{attribute 'monitoring':='call'}
PROPERTY MoversInZone : REFERENCE TO ARRAY [0..(CHALET_BaseComponents.BaseParameterlist.MAX_OBJECTS-1)] OF I_XP_Mover_PLC // Return a sorted list of movers in this zone. Index 0 is the mover in Front.
GET
END_GET
END_PROPERTY

END_INTERFACE

// COMPONENTs/Path/FB_XP_Path
{attribute 'enable_dynamic_creation'}
{attribute 'no_explicit_call' := 'Do not call the body - Stick to OOP'}
FUNCTION_BLOCK FB_XP_Path EXTENDS FB_CH_Object IMPLEMENTS I_XP_Path
VAR
	fbTracksUsed : FB_CH_List;
	ipStartStation, ipDestinationStation : I_XP_Station;
	fPathLength : LREAL;
END_VAR

METHOD DistanceToDestiantion : LREAL
VAR_INPUT
	ipTrack : I_XP_Track;
	fPosOnTrack : LREAL;
END_VAR
VAR
	bCorrectPos, bCorrectTrack : BOOL;
	bPosFound : BOOL;
	fDistReturnNotOnThisTrack : LREAL;
	fStart, fEnd : LREAL;
	ipEachTrack : I_XP_Track; 
END_VAR
VAR
	//Todo add tolerance to Size >1
	fToleranceWindow : LREAL := 0.001;//[mm] if Mover is this distance mor far away from the parent, return 0mm
END_VAR
IF ipTrack = 0 THEN
	//Error -  invalide interface
	DistanceToDestiantion := CHALET_BaseComponents.GVL_Datatypes.cMaxLreal;
	RETURN;
END_IF

fDistReturnNotOnThisTrack := CHALET_BaseComponents.GVL_Datatypes.cMaxLreal;

IF (fbTracksUsed.OIDInList(ipTrack.OID) = 0) OR fPosOnTrack < 0 OR  fPosOnTrack > ipTrack.Length THEN
	//Error -  position not on track
	DistanceToDestiantion := fDistReturnNotOnThisTrack;
	RETURN;
END_IF


IF fbTracksUsed.Size = 1 THEN
	bCorrectPos := F_InLimitTest(fMinimum :=  THIS^.StationStart.PositionOnTrack, fInput:=fPosOnTrack , fMaximum:=  (THIS^.StationDestination.PositionOnTrack + fToleranceWindow));
	bCorrectTrack := (ipTrack = StationDestination.AccocietedTrack);

	IF bCorrectPos AND bCorrectTrack THEN
		DistanceToDestiantion := F_GetDistToPosModulo(fTargetPosition := THIS^.StationDestination.PositionOnTrack, fActualPosition := fPosOnTrack, fModulo := ipTrack.Length);
		//check tolerance window
		IF (DistanceToDestiantion + fToleranceWindow) >= ipTrack.Length THEN
			DistanceToDestiantion := 0.0;
		END_IF
	ELSE
		DistanceToDestiantion := fDistReturnNotOnThisTrack;
	END_IF
	RETURN;
END_IF


IF fbTracksUsed.Size > 1 THEN 
	fbTracksUsed.ResetIterator();	
	
	////First track in list
	IF ToXpTrack(fbTracksUsed.GetNextObject(),ipEachTrack) THEN
		fStart 	:= THIS^.StationStart.PositionOnTrack;
		fEnd 	:= ipEachTrack.Length;
		
		bCorrectPos := F_InLimitTest(fMinimum :=  fStart, fInput:=fPosOnTrack , fMaximum:=  fEnd);
		bCorrectTrack := (ipTrack = ipEachTrack);
		IF bCorrectPos AND bCorrectTrack THEN
			bPosFound := TRUE;
			DistanceToDestiantion := fEnd - fPosOnTrack;
		END_IF
	END_IF
	
	
	//All tracks in between
	WHILE fbTracksUsed.HasNextObject() DO
		IF ToXpTrack(fbTracksUsed.GetNextObject(),ipEachTrack) AND_THEN fbTracksUsed.HasNextObject() THEN
			fStart 	:= 0;
			fEnd 	:= ipEachTrack.Length;
			
			// still locking for the startpoint to measure the distance to Destination
			IF NOT bPosFound THEN
				bCorrectPos := F_InLimitTest(fMinimum :=  fStart, fInput:=fPosOnTrack , fMaximum:=  fEnd);
				bCorrectTrack := (ipTrack = ipEachTrack);
				IF bCorrectPos AND bCorrectTrack THEN
					bPosFound := TRUE;
					DistanceToDestiantion := fEnd - fPosOnTrack;
				END_IF
			ELSE
				// add all the tracklengths
				DistanceToDestiantion := DistanceToDestiantion + fEnd;		
			END_IF
		END_IF
	END_WHILE	
	
	
	//Last track
		fStart 	:= 0;
		fEnd 	:= (THIS^.StationDestination.PositionOnTrack + fToleranceWindow);
		// still locking for the startpoint to measure the distance to Destination
		IF NOT bPosFound THEN
			bCorrectPos := F_InLimitTest(fMinimum :=  fStart, fInput:=fPosOnTrack , fMaximum :=  fEnd);
			bCorrectTrack := (ipTrack = ipEachTrack);
			IF bCorrectPos AND bCorrectTrack THEN
				bPosFound := TRUE;
				DistanceToDestiantion := MAX(0, THIS^.StationDestination.PositionOnTrack - fPosOnTrack);
			END_IF
		ELSE
			// add all the tracklengths
			DistanceToDestiantion := DistanceToDestiantion + fEnd;		
		END_IF

	
	fbTracksUsed.RestoreIterator();
	
	IF NOT bPosFound THEN
		DistanceToDestiantion := fDistReturnNotOnThisTrack;
		RETURN;
	END_IF
END_IF
END_METHOD

{attribute 'monitoring':='call'}
//[mm]
PROPERTY Length : LREAL
GET
Length := THIS^.fPathLength;
END_GET
SET
THIS^.fPathLength := Length;
END_SET
END_PROPERTY

{attribute 'monitoring':='call'}
PROPERTY LUID : STRING //Locally unique identifier
GET
VAR
	sTempName : STRING;
END_VAR
IF ipStartStation <> 0 AND ipDestinationStation <> 0 THEN
	sTempName := CONCAT(sTempName, ipStartStation.LUID);
	sTempName := CONCAT(sTempName, ' to ' );
	sTempName := CONCAT(sTempName, ipDestinationStation.LUID);
	
ELSIF ipStartStation <> 0 THEN
	sTempName := CONCAT(sTempName, ipStartStation.LUID);
	sTempName := CONCAT(sTempName, ' to ?' );

ELSIF ipDestinationStation <> 0 THEN
	sTempName := CONCAT(sTempName, '? to ' );
	sTempName := CONCAT(sTempName, ipDestinationStation.LUID);
	
ELSE 
	sTempName := ' Unknown path';
END_IF


LUID := sTempName;
END_GET
END_PROPERTY

{attribute 'monitoring':='call'}
PROPERTY StationDestination : I_XP_Station
GET
StationDestination := THIS^.ipDestinationStation;
END_GET
SET
THIS^.ipDestinationStation := StationDestination;
END_SET
END_PROPERTY

{attribute 'monitoring':='call'}
PROPERTY StationStart  : I_XP_Station
GET
StationStart := THIS^.ipStartStation;
END_GET
SET
THIS^.ipStartStation := StationStart;
END_SET
END_PROPERTY

{attribute 'monitoring':='call'}
//List of tracks
PROPERTY TracksUsed : REFERENCE TO FB_CH_List
GET
TracksUsed REF= THIS^.fbTracksUsed;
END_GET
END_PROPERTY

END_FUNCTION_BLOCK

// FUNCTIONs/F_InLimitTest
FUNCTION F_InLimitTest : BOOL
VAR_INPUT
	fMinimum 	: LREAL;
	fMaximum 	: LREAL;
	fInput 		: LREAL;
END_VAR

//Normal case
// 9 Max
// 5 Test
// 1 Min
IF fMinimum <= fMaximum THEN
	F_InLimitTest := (fInput >= fMinimum) AND (fInput <= fMaximum);
	
//Modulo case	
// 6 | 6  Max
// 5 | 9  Test
// 8 | 8  Min
ELSIF fMinimum > fMaximum THEN
	F_InLimitTest := NOT((fInput > fMaximum) AND (fInput < fMinimum));
END_IF

END_FUNCTION

// FUNCTIONs/F_GetDistToPosModulo
FUNCTION F_GetDistToPosModulo : LREAL //This is only working in Positiv Direktion
VAR_INPUT
	fTargetPosition : LREAL;
	fActualPosition : LREAL;
	fModulo 		: LREAL;
END_VAR

VAR

END_VAR

IF fTargetPosition < fActualPosition THEN
	fTargetPosition := fTargetPosition + fModulo;
END_IF

F_GetDistToPosModulo := fTargetPosition - fActualPosition;

END_FUNCTION

// COMPONENTs/Stationen/A-Star-Node/FB_AStarNode
FUNCTION_BLOCK FB_AStarNode EXTENDS FB_CH_Object IMPLEMENTS I_PathAStarNode
VAR
	{attribute 'hide'}  
	ipStation : I_XP_Station;
	{attribute 'hide'}  
	fbRouteUsedToNode : FB_CH_LIST;	
END_VAR

{attribute 'monitoring':='call'}
PROPERTY LUID : STRING
GET
IF THIS^.Station <> 0 THEN
	LUID := THIS^.Station.LUID;
END_IF
END_GET
END_PROPERTY

{attribute 'monitoring':='call'}
PROPERTY PathLength : LREAL
GET
VAR
	ipEachPath : I_XP_Path;
END_VAR
PathLength := 0.0;


fbRouteUsedToNode.ResetIterator();
WHILE fbRouteUsedToNode.HasNextObject() DO
	IF __QUERYINTERFACE(fbRouteUsedToNode.GetNextObject(), ipEachPath) THEN
		PathLength := PathLength + ipEachPath.Length;
	END_IF
END_WHILE
fbRouteUsedToNode.RestoreIterator();
END_GET
END_PROPERTY

{attribute 'monitoring':='call'}
PROPERTY RouteUsedToNode : REFERENCE TO FB_CH_List
GET
RouteUsedToNode REF= fbRouteUsedToNode;
END_GET
END_PROPERTY

//here in this case the SortOrder is used to get the shortest path. 
PROPERTY SortOrderInList : UDINT
GET
SortOrderInList := TO_UDINT(THIS^.PathLength);
END_GET
END_PROPERTY

{attribute 'monitoring':='call'}
PROPERTY Station : I_XP_Station
GET
Station := ipStation;
END_GET
SET
ipStation := Station;
END_SET
END_PROPERTY

END_FUNCTION_BLOCK

// COMPONENTs/Stationen/A-Star-Node/I_PathAStarNode
INTERFACE I_PathAStarNode EXTENDS I_CH_Object

{attribute 'monitoring':='call'}
PROPERTY PathLength : LREAL
GET
END_GET
END_PROPERTY

{attribute 'monitoring':='call'}
PROPERTY RouteUsedToNode : REFERENCE TO FB_CH_List
GET
END_GET
END_PROPERTY

{attribute 'monitoring':='call'}
PROPERTY Station : I_XP_Station
GET
END_GET
SET
END_SET
END_PROPERTY

END_INTERFACE

// COMPONENTs/Stationen/FB_XP_Station
{attribute 'enable_dynamic_creation'}
{attribute 'no_explicit_call' := 'Do not call the body - Stick to OOP'}
(* XPlanar station - n per associated XPlanar. Can be instantiated as an array and/or individually
	The stations are the main component of the application. As soon as the system has been started up and all movers are on the track, the movers are only sent from one station to the next.
	Parameters:
		xPos, yPos 			= Absolute position of the station on the xPlanar.
		ipAccocietedTrack 	= The track on which the station is located. If the XY position is not on this track, the next possible track position is assumed on this track.
		sUniqueName 		= Unique name that may only exist once.
		sTargetGroup 		= A name for a group to which this station belongs. Important for redundant stations
 *)	
FUNCTION_BLOCK FB_XP_Station EXTENDS FB_CH_Object IMPLEMENTS I_XP_Station, I_XP_Station_PLC
VAR
	//optional - To visualize the station position in LiveView
	fbOptionalTrackUsedInLiveView : MC_PlanarTrack;

	{attribute 'hide'}
	bErrorDuringFbInit : BOOL;	//Fatal error - Not possible to reset
	
	{attribute 'hide'}
	bInitDone : BOOL;
	{attribute 'hide'}	
	bTrackIsSetInFbInit : BOOL;
	{attribute 'hide'}	
	bMoversInPlace : BOOL;
	{attribute 'hide'}                   	
	eActiveCommand 		: CHALET_Nc.E_NcAxisCommands := CHALET_Nc.E_NcAxisCommands.None;
	{attribute 'hide'}	
	ipXpSystem : I_XP_System_Registration;
	{attribute 'hide'}
	bReadyToRecvMovers 		: BOOL := TRUE;
	{attribute 'hide'}
	nCtsMoversMustLeaveThisStation : UDINT;
	{attribute 'hide'}
	sTargetGroup 				: STRING;
	
	{attribute 'hide'}
	bSuppressDynamicsChange		: BOOL; // Suppress to change the dynamic(Gap+velocity) of passing movers. This is usefull in startup
	{attribute 'hide'}
	fMoverGapAtExit 			: LREAL := XPlanarParameterlist.F_GAP_DEFAULT; // Every mover that leaves or passes the station gets this new gap as a target.
	{attribute 'hide'}	
	fbPositionPlanned : PositionXY; //this is the configured/planned position of the station. set via FB_init. If it is not on the track, the PosOnTrackXY is different
	{attribute 'hide'}	
	fPositionOnTrack : LREAL;
	{attribute 'hide'}
	fbPositionOnTrackXY : PositionXY;	
	{attribute 'hide'}	
	nState_Configuring: INT;
	{attribute 'hide'}	
	ipAccocietedTrack : I_XP_Track;
	{attribute 'hide'}
	nMoverQueueSize 			: UINT;
	{attribute 'hide'}
	fTargetPosWindow			: LREAL := 0.05; //[mm]
	{attribute 'hide'}
	tTargetPosMonitoringTime	: TIME := T#0MS;

	
	(*List of stations*)
	{attribute 'hide'}	
	fbStationsAhead : FB_CH_List;
	{attribute 'hide'}	
	fbStationsBehinde : FB_CH_List;
	
	(*List of paths*)
	{attribute 'hide'}	
	fbListPathAhead : FB_CH_List;
	{attribute 'hide'}
	fbListPathBehind : FB_CH_List;
	
	(* Lists to handle the ownership of movers *)
	{attribute 'hide'}
	fbAssignedMovers 			: FB_CH_List;		// Movers approaching the station. This station is the parent of this movers
	{attribute 'hide'}
	fbFeedback : FB_CH_Feedback(ipSourceInfo := fbSourceInfo);		
	
	//Simulation
	{attribute 'hide'}
	fSimulationProcessDuration 	: LREAL; //[s]
	{attribute 'hide'}
	sSimulationTargetStation	: STRING; //GroupID of the target station to automatic send after the duration
	
	
	//ipXpSystem Is Not Valid at this point, call the konstruktor again in the FB_Init
	{attribute 'hide'}
	fbTrigger 					: FB_XP_Trigger(ipXpSystem);
	{attribute 'hide'}
	fbSortedListMoversInQueue	: FB_XP_SoretedListOfMover(	ipXpStation := THIS^,
															ipListOfMoversToCheck := fbAssignedMovers );
	{attribute 'hide'}
	fDecisionDistance: LREAL;//[mm]
	{attribute 'hide'}
	bNetworkHasTrackBranches : BOOL;//True if atleas on branche is existing in network
	{attribute 'hide'}
	sFilter : STRING :=  XPlanarParameterlist.S_ANY_STATION_NAME;
	{attribute 'hide'}	
	fbAlarmStationIsBlocked : FB_TcAlarm;
END_VAR

// Dynamic to use if an Mvoer passes the station
// Every mover that leaves or passes the station gets this new velo as a target.
VAR
	{attribute 'hide'}	
	fMoverVeloAtExit : MC_LREAL := MC_DEFAULT; //equivalent to data type LREAL + MC_DEFAULT, MC_MAXIMUM
	{attribute 'hide'}	
    fMoverAccAtExit : MC_LREAL := MC_DEFAULT; //equivalent to data type LREAL + MC_DEFAULT, MC_MAXIMUM
	{attribute 'hide'}	
    fMoverDecAtExit : MC_LREAL := MC_DEFAULT; //equivalent to data type LREAL + MC_DEFAULT, MC_MAXIMUM
END_VAR

METHOD PROTECTED CheckInvalideParameter : HRESULT
VAR
 	ipStation : I_XP_Station;
	fbListOfStationsToCheck : FB_CH_List;
END_VAR
VAR_INST
	{attribute 'hide'}	
	fbAlarm : FB_TcAlarm;
END_VAR
//Get a list of all station whitout this station
fbListOfStationsToCheck.Duplicate(THIS^.ipXpSystem.StationsUsed);
fbListOfStationsToCheck.RemoveObject(THIS^);


fbListOfStationsToCheck.ResetIterator();
WHILE fbListOfStationsToCheck.HasNextObject() DO
	IF ToXpStation(fbListOfStationsToCheck.GetNextObject(), ipStation) THEN
		
		//Check for same positions
		IF (ipStation.PositionOnTrack = THIS^.PositionOnTrack) AND (ipStation.AccocietedTrack = THIS^.AccocietedTrack)  THEN
			//Error two stations have same position on track
			CheckInvalideParameter := E_FAIL;
			IF NOT fbAlarm.bRaised THEN
				fbAlarm.CreateEx(stEventEntry:=TC_EVENTS.CHALET_XPlanar_Events.DuplicateStationPositions, ipSourceInfo := THIS^.fbSourceInfo, bWithConfirmation := FALSE);
				fbAlarm.ipArguments.AddStringByValue(THIS^.LUID).AddStringByValue(ipStation.LUID);
				fbAlarm.Raise(0);			
			END_IF
			RETURN;
		END_IF
		
		//Check same unique id
		IF (ipStation.LUID = THIS^.LUID) THEN
			//Error two stations have same unique id
			CheckInvalideParameter := E_FAIL;
			IF NOT fbAlarm.bRaised THEN
				fbAlarm.CreateEx(stEventEntry:=TC_EVENTS.CHALET_XPlanar_Events.DuplicateStationName, ipSourceInfo := THIS^.fbSourceInfo, bWithConfirmation := FALSE);
				fbAlarm.ipArguments.AddStringByValue(THIS^.LUID);
				fbAlarm.Raise(0);			
			END_IF
			RETURN;
		END_IF
		
		fbListOfStationsToCheck.RemoveObject(ipStation);
	END_IF
END_WHILE
END_METHOD

METHOD protected GetAccocietedTrack : HRESULT
VAR
	ipTrack : I_XP_Track;

	fPosOnTrack, fDist	: LREAL;
	fbPositionXYC : PositionXYC;
	fbPositionXY : PositionXY;
	ipClosestTrack : I_XP_Track;
	fDistClosestTrack : LREAL := CHALET_BaseComponents.GVL_Datatypes.cMaxLreal;
END_VAR
//If track is not defind during FB_init, get closest track 
IF NOT bTrackIsSetInFbInit THEN
	THIS^.ipAccocietedTrack := 0;
	THIS^.ipXpSystem.Tracks.ResetIterator();
	WHILE THIS^.ipXpSystem.Tracks.HasNextObject() DO
		IF ToXpTrack(THIS^.ipXpSystem.Tracks.GetNextObject(),ipTrack) THEN 
			
			fPosOnTrack := ipTrack.PlanarTrack.GetArcLengthClosestTo(geometry:= THIS^.fbPositionPlanned);
			//Get the XYC Pos on track
			ipTrack.PlanarTrack.GetPositionAt(fPosOnTrack, fbPositionXYC);
			//Get radius/ distance to positionTarget
			fbPositionXY.x  := THIS^.fbPositionPlanned.x - fbPositionXYC.x;
			fbPositionXY.y  := THIS^.fbPositionPlanned.y - fbPositionXYC.y;
			fDist := fbPositionXY.GetRadius();
			
			IF fDist < fDistClosestTrack THEN
				fDistClosestTrack := fDist;
				ipClosestTrack := ipTrack;
			END_IF
		END_IF
	END_WHILE
	THIS^.ipXpSystem.Tracks.RestoreIterator();
	
	
	THIS^.ipAccocietedTrack := ipClosestTrack;	
END_IF

// Error - No track found
IF THIS^.ipAccocietedTrack = 0 THEN
	GetAccocietedTrack := E_FAIL;
	RETURN;
END_IF
END_METHOD

METHOD GetDecisionDistance : HRESULT
VAR
	fDistToStartOfTrack : LREAL := CHALET_BaseComponents.GVL_Datatypes.cMaxLreal;
	fDistStationBehind : LREAL := CHALET_BaseComponents.GVL_Datatypes.cMaxLreal;
	
	ipPath : I_XP_Path;
END_VAR
(*
As soon as the mover is closer than this distance, the mover can be sent on to the next one if necessary.
This is the distance from the station to the end of the track or the shortest path to this station. Depending on which is closer. This is to ensure that the mover can no longer be overhauled.
*)
fDistToStartOfTrack := THIS^.PositionOnTrack;

THIS^.PathsBehinde.ResetIterator();
WHILE THIS^.PathsBehinde.HasNextObject() DO
	IF __QUERYINTERFACE(THIS^.PathsBehinde.GetNextObject(), ipPath) THEN
		fDistStationBehind := MIN(fDistStationBehind, ipPath.Length);
	END_IF
END_WHILE
THIS^.PathsBehinde.RestoreIterator();

THIS^.fDecisionDistance := CHALET_BaseComponents.GVL_Datatypes.cMaxLreal;
THIS^.fDecisionDistance := MIN(THIS^.fDecisionDistance, (fDistToStartOfTrack - 1.0));
THIS^.fDecisionDistance := MIN(THIS^.fDecisionDistance, (fDistStationBehind - 1.0));
THIS^.fDecisionDistance := MIN(THIS^.fDecisionDistance, XPlanarParameterlist.F_DIST_SET_NEW_MOVE_CMD_BEFORE_REACHING_PARENT_STATION);


IF THIS^.fDecisionDistance < 1.0 THEN 
	THIS^.fDecisionDistance := 1.0;
END_IF

GetDecisionDistance := S_OK;
END_METHOD

METHOD protected GetPathsAhead : HRESULT
VAR_INPUT
END_VAR

VAR
	fbPathElementsToCheck : FB_CH_List;
	fbListStationsToGetClosest : FB_CH_List;	
	ipObjectPathAhead 				: I_CH_Object;
	ipStation,ipStation1,ipStation2 	: I_XP_Station;
	ipTrack					: I_XP_Track; 
	ipLastAddedTrack 		: I_XP_Track;
	ipPath 					: I_XP_Path;
	ipPathCurrentLoop  		: I_XP_Path;
	
	
	pFbPath, pFbPathCurrentLoop : POINTER TO FB_XP_Path;
	
	fSeachStartPoint : LREAL;
	nIdx : UDINT;
END_VAR
(*
Check whether there is a station further ahead on this track than this one.
If there is no other station on the track, the previous tracks are filled into a list and searched one after the other to see if they have valid stations. 
If the tracks also have no stations, the track before it is added to the list,...
*)

//Clear list, delete dynamic_creation path objects
WHILE NOT fbListPathAhead.IsEmpty DO
	ipObjectPathAhead := fbListPathAhead.GetRandomObject();
	fbListPathAhead.RemoveObject(ipObjectPathAhead);
	
	//get pointer and delete
	IF __QUERYPOINTER(ipObjectPathAhead, pFbPath) THEN
		__DELETE(pFbPath);
	END_IF	
		
END_WHILE


//new dynamic_creation path objects
pFbPath := __NEW(FB_XP_Path);
//init path
pFbPath^.StationStart := THIS^;
pFbPath^.TracksUsed.ResetIterator();
pFbPath^.TracksUsed.AddObject(THIS^.AccocietedTrack);

//add to list
fbPathElementsToCheck.AddObject(pFbPath^);

//On first pathsearch get an Station who is further ahead than this
fSeachStartPoint := THIS^.PositionOnTrack;



//While list is not empty
WHILE NOT fbPathElementsToCheck.IsEmpty DO
	__QUERYINTERFACE(fbPathElementsToCheck.GetRandomObject(), ipPathCurrentLoop);
	__QUERYINTERFACE(ipPathCurrentLoop.TracksUsed.GetNextObject(),ipLastAddedTrack);
	
	
	//Closed loop
	IF ipLastAddedTrack.ClosedLoop THEN
		//on closed-loop add all stations of this track to list
		fbListStationsToGetClosest.Duplicate(ipLastAddedTrack.StationsOnTrack);
	
		//remove THIS station from list if more than on station is existing
		IF fbListStationsToGetClosest.Size > 1 THEN
			fbListStationsToGetClosest.RemoveObject(THIS^);
		END_IF
	
		
	
	ELSE
		//Not closed loop	
		//Get a List of all stations on track Position > Startpoint
		ipLastAddedTrack.StationsOnTrack.ResetIterator();
		fbListStationsToGetClosest.Clear();
		WHILE ipLastAddedTrack.StationsOnTrack.HasNextObject() DO
			IF ToXpStation(ipLastAddedTrack.StationsOnTrack.GetNextObject(),ipStation) THEN
				//Add all station ahead to list. on closed-loop add all stations of this track to list
				IF ipStation.PositionOnTrack > fSeachStartPoint THEN
					fbListStationsToGetClosest.AddObject(ipStation);
				END_IF
			END_IF
		END_WHILE	
	END_IF
		
	

	
	//Get closest to startpos(0mm)
	WHILE fbListStationsToGetClosest.Size > 1 DO
		fbListStationsToGetClosest.ResetIterator();
		__QUERYINTERFACE(fbListStationsToGetClosest.GetNextObject(),ipStation1);
		__QUERYINTERFACE(fbListStationsToGetClosest.GetNextObject(),ipStation2);
		
		//If station1 is closer to start than station2, remove station2
		IF 		F_GetDistToPosModulo(fTargetPosition := ipStation1.PositionOnTrack, fActualPosition := fSeachStartPoint, fModulo := ipLastAddedTrack.Length) 
			< 	F_GetDistToPosModulo(fTargetPosition := ipStation2.PositionOnTrack, fActualPosition := fSeachStartPoint, fModulo := ipLastAddedTrack.Length) THEN
			fbListStationsToGetClosest.RemoveObject(ipStation2);
		ELSE	
			fbListStationsToGetClosest.RemoveObject(ipStation1);
		END_IF
	END_WHILE
	
	
	IF fbListStationsToGetClosest.Size = 1 THEN
		//Station FOUND
		__QUERYINTERFACE(fbListStationsToGetClosest.GetRandomObject(), ipStation);
		ipPathCurrentLoop.StationDestination := ipStation;
		
		//Calculate Tracklentgh
		ipPathCurrentLoop.TracksUsed.ResetIterator();
		WHILE ipPathCurrentLoop.TracksUsed.HasNextObject() DO
			IF ToXpTrack(ipPathCurrentLoop.TracksUsed.GetNextObject(),ipTrack) THEN
				ipPathCurrentLoop.Length := ipPathCurrentLoop.Length + ipTrack.Length;
			END_IF
		END_WHILE	
		ipPathCurrentLoop.Length := ipPathCurrentLoop.Length - ipPathCurrentLoop.StationStart.PositionOnTrack;
		ipPathCurrentLoop.Length := ipPathCurrentLoop.Length - ipPathCurrentLoop.StationDestination.AccocietedTrack.Length + ipPathCurrentLoop.StationDestination.PositionOnTrack;
		
		//Modulo on cloosed track add 1 track length 
		IF ipPathCurrentLoop.StationStart.AccocietedTrack = ipPathCurrentLoop.StationDestination.AccocietedTrack AND 
			ipPathCurrentLoop.StationStart.PositionOnTrack > ipPathCurrentLoop.StationDestination.PositionOnTrack THEN
				ipPathCurrentLoop.Length := ipPathCurrentLoop.Length + ipPathCurrentLoop.StationDestination.AccocietedTrack.Length;
		END_IF
		
		fbListPathAhead.AddObject(ipPathCurrentLoop);
		fbPathElementsToCheck.RemoveObject(ipPathCurrentLoop);
	ELSE
		//Station NOT-FOUND, add the subsequent tracks in the list
		ipLastAddedTrack.TracksAhead.ResetIterator();
		WHILE ipLastAddedTrack.TracksAhead.HasNextObject() DO
			ToXpTrack(ipLastAddedTrack.TracksAhead.GetNextObject(), ipTrack);
			//dublicate current path
			pFbPath := __NEW(FB_XP_Path);
			//Get pointer from fb behinde this interface
			__QUERYPOINTER(ipPathCurrentLoop, pFbPathCurrentLoop);
			MEMCPY(destAddr := pFbPath, srcAddr := pFbPathCurrentLoop, n := SIZEOF(FB_XP_Path));
			//Add the new track to fresh created path
			pFbPath^.TracksUsed.AddObject(ipTrack);
			//Add to list to check
			fbPathElementsToCheck.AddObject(pFbPath^);
			
		END_WHILE

		
		//delete current path
		fbPathElementsToCheck.RemoveObject(ipPathCurrentLoop);

		//get pointer and delete
		IF __QUERYPOINTER(ipPathCurrentLoop, pFbPath) THEN
			__DELETE(pFbPath);
		END_IF	
		
	END_IF

	fSeachStartPoint := -0.1;
END_WHILE
END_METHOD

METHOD protected GetPathsBehind : HRESULT
VAR
	ipThisStation : I_XP_Station;
	ipXpStation : I_XP_Station;
	ipPath		: I_XP_Path;
END_VAR
ipThisStation := THIS^;
fbListPathBehind.Clear();

THIS^.fbStationsBehinde.ResetIterator();
WHILE THIS^.fbStationsBehinde.HasNextObject() DO
	IF __QUERYINTERFACE(THIS^.fbStationsBehinde.GetNextObject(),ipXpStation) THEN
		ipXpStation.PathsAhead.ResetIterator();
		WHILE ipXpStation.PathsAhead.HasNextObject() DO
			IF __QUERYINTERFACE(ipXpStation.PathsAhead.GetNextObject(),ipPath) AND_THEN ipPath.StationDestination = ipThisStation THEN
				//add path to this station to list
				fbListPathBehind.AddObject(ipPath);
			END_IF
		END_WHILE	
	END_IF
END_WHILE
END_METHOD

METHOD PROTECTED GetPosOnTrack : HRESULT
VAR
	fbPositionXYC : PositionXYC;
END_VAR
//GetArcLengthClosestTo track
THIS^.fPositionOnTrack := THIS^.ipAccocietedTrack.PlanarTrack.GetArcLengthClosestTo(geometry:= THIS^.fbPositionPlanned);

//Get the XYC Pos on track
THIS^.ipAccocietedTrack.PlanarTrack.GetPositionAt(THIS^.PositionOnTrack, fbPositionXYC);

//XYC -> XY
THIS^.fbPositionOnTrackXY.SetValuesXY(fbPositionXYC.x,fbPositionXYC.y);


//Check for NaN
IF NOT(THIS^.fPositionOnTrack = THIS^.fPositionOnTrack) THEN
	GetPosOnTrack := E_FAIL;
	RETURN;
END_IF
END_METHOD

METHOD PROTECTED GetStationAhead : HRESULT
VAR
	ipPath 		: I_XP_Path;
END_VAR
fbStationsAhead.Clear();


fbListPathAhead.ResetIterator();
WHILE fbListPathAhead.HasNextObject() DO
	IF __QUERYINTERFACE(fbListPathAhead.GetNextObject(),ipPath) THEN
		//add StationDestination to list
		fbStationsAhead.AddObject(ipPath.StationDestination);
	END_IF
END_WHILE
END_METHOD

METHOD PROTECTED GetStationBehinde : HRESULT
VAR_INPUT
END_VAR
VAR
	ipThisStation : I_XP_Station;
	ipXpStation : I_XP_Station;
	ipXpStationAhead : I_XP_Station;
END_VAR
ipThisStation := THIS^;
fbStationsBehinde.Clear();

//Check each Station
THIS^.ipXpSystem.StationsUsed.ResetIterator();
WHILE THIS^.ipXpSystem.StationsUsed.HasNextObject() DO
	IF __QUERYINTERFACE(THIS^.ipXpSystem.StationsUsed.GetNextObject(),ipXpStation) THEN
		//check the list of stations ahead if this station one is existing
		ipXpStation.StationsAhead.ResetIterator();
		WHILE ipXpStation.StationsAhead.HasNextObject() DO
			IF __QUERYINTERFACE(ipXpStation.StationsAhead.GetNextObject(),ipXpStationAhead) AND_THEN (ipXpStationAhead = ipThisStation) THEN
				//add station to list
				fbStationsBehinde.AddObject(ipXpStation);
			END_IF
		END_WHILE	
	END_IF
END_WHILE	
THIS^.ipXpSystem.StationsUsed.RestoreIterator();
END_METHOD

METHOD PROTECTED ManageAutomaticallyGeneratedStations : HRESULT
VAR
	ipThisStation : I_XP_Station := THIS^;
	ipTempTrackAhead : I_XP_Track;
	bThisStationIsCreatedAutomatically : BOOL;
	
	bOtherStationsOnThisTrack : BOOL;
	bAnotherTrackAhed : BOOL;
	
	pfbListAllUsedStations : POINTER TO FB_CH_List;
END_VAR
// Check if this station was created by the user, e.g., as a process station, or if it was created automatically at the end of the track to improve track management.
bThisStationIsCreatedAutomatically := (ipThisStation = THIS^.AccocietedTrack.HelperStationAtEndOfTrack);

// Only check automaticali created stations
IF NOT bThisStationIsCreatedAutomatically THEN
	ManageAutomaticallyGeneratedStations := S_OK;
	RETURN;
END_IF



//Set position of this automatic generated station to the end of the accocieted Track
THIS^.PositionXY.x := THIS^.AccocietedTrack.EndPosition.x;
THIS^.PositionXY.y := THIS^.AccocietedTrack.EndPosition.y;



//Check if other Stations are existiong on this track
IF THIS^.AccocietedTrack.StationsOnTrack.Size > 1 THEN
	bOtherStationsOnThisTrack := TRUE;
END_IF

//Another track is before this accocieted track. But the track in front of me is only allowed to have this one track in behind of it.
__QUERYINTERFACE(THIS^.AccocietedTrack.TracksAhead.GetRandomObject(), ipTempTrackAhead);
IF ipTempTrackAhead <> 0 AND_THEN ipTempTrackAhead.TracksBehinde.Size = 1 THEN
	bAnotherTrackAhed := TRUE;
END_IF

//Remove this station from list
/// Todo remove Querypointer - not very OOP
IF (bOtherStationsOnThisTrack OR bAnotherTrackAhed OR NOT XPlanarParameterlist.B_AUTOMATIC_GENARATE_HELPER_STATIONS ) AND __QUERYPOINTER(THIS^.ipXpSystem.StationsUsed, pfbListAllUsedStations) THEN
	//Remove single trackpoint if station is not used
	THIS^.fbOptionalTrackUsedInLiveView.Clear(0);
	pfbListAllUsedStations^.RemoveObject(THIS^);
END_IF
END_METHOD

METHOD SetTrackObjName : HRESULT
VAR
	ipComObject : ITComObject;
	sName : STRING;
END_VAR
FW_ObjMgr_GetObjectInstance(oid:= THIS^.fbOptionalTrackUsedInLiveView.MCTOPLC_STD.TrackOID, iid:= TC_GLOBAL_IID_LIST.IID_ITComObject, pipUnk:= ADR(ipComObject));
IF ipComObject <> 0 THEN
	sName := THIS^.LUID;
	ipComObject.TcSetObjectName(ADR(sName));
	FW_SafeRelease(ADR(ipComObject));
END_IF
END_METHOD

//Call this Methode whith seq 0->99, and wait each step until S_OK is returned
METHOD Configure : HRESULT
VAR_INPUT
	nSeq : UINT; //0->100
END_VAR

VAR_INST
	{attribute 'hide'}
	fbFeedback : MC_PlanarFeedback;	
END_VAR
VAR
	bOptionalTrackUsedInLiveViewIsMapped : BOOL;
	fbPositionXYC : PositionXYC;
	ipEachTrack : I_XP_Track;
END_VAR
bOptionalTrackUsedInLiveViewIsMapped := fbOptionalTrackUsedInLiveView.MCTOPLC_STD.TrackOID <> 0;

CASE nSeq OF
	5:	//Get interface of trackobject
		Configure := THIS^.GetAccocietedTrack();	

	10: //Get closest XY-Position on track
		Configure := THIS^.GetPosOnTrack();
		
	11:	//Automatic add/remove this station from list of all station if it is createt automatic at the end of each track and is (not) used	
		Configure := THIS^.ManageAutomaticallyGeneratedStations();
		
	12: //Check id is unique and not multiple stations at same position
		Configure := THIS^.CheckInvalideParameter();		
				
	13:	//Init Tigger
		fbTrigger.AccocietedTrack := THIS^.AccocietedTrack;
		fbTrigger.PositionOnTrack := THIS^.PositionOnTrack;
		fbTrigger.ListOfMoversToCheck := THIS^.ipXpSystem.MoversPresent;//All mover
		fbTrigger.TriggerDirection := Tc3_Mc3Definitions. MC_DIRECTION.mcDirectionPositive;
		Configure := fbTrigger.Initialize();
	
	14:	//Init Zone		
		Configure := fbSortedListMoversInQueue.Initialize();	
	
	20: //Fill the list of all paths before this station
		Configure := THIS^.GetPathsAhead();		
		
	25: //Fill the list of all stations before this station
		Configure := THIS^.GetStationAhead();

	30: //Fill the list of all paths behinde this station
		Configure := THIS^.GetStationBehinde();	
			
	35: //Fill the list of all stations behinde this station
		Configure := THIS^.GetPathsBehind();

	40: //Determine the distance from which the station can give a new command to a mover
		Configure := THIS^.GetDecisionDistance();
		

//----------------------------------------------------------------		
//The station can optionally be linked to a track object. this track is then displayed in the live view.
//It takes several cycles to prepare the object
	80: IF bOptionalTrackUsedInLiveViewIsMapped THEN
			fbOptionalTrackUsedInLiveView.Clear(fbFeedback);
		END_IF
		
	81:	//Wait for clearing
		IF bOptionalTrackUsedInLiveViewIsMapped THEN
			IF fbFeedback.Done THEN
				Configure := S_OK;
			ELSIF fbFeedback.Busy THEN
				Configure := S_PENDING;
			ELSIF fbFeedback.Error THEN
				Configure := E_FAIL;
			END_IF	
		END_IF

	82: //Set position 
		IF bOptionalTrackUsedInLiveViewIsMapped THEN
			fbPositionXYC.SetValuesXY(THIS^.PositionOnTrackXY.x, THIS^.PositionOnTrackXY.y);
			fbOptionalTrackUsedInLiveView.AppendPosition(position := fbPositionXYC, commandFeedback:= fbFeedback);	
		END_IF	
	
	83:	//Wait for set position
		IF bOptionalTrackUsedInLiveViewIsMapped THEN
			IF fbFeedback.Done THEN
				Configure := S_OK;
			ELSIF fbFeedback.Busy THEN
				Configure := S_PENDING;
			ELSIF fbFeedback.Error THEN
				Configure := E_FAIL;
			END_IF	
		END_IF
		
	84:	//Set name of "track" to stationsname 
		IF bOptionalTrackUsedInLiveViewIsMapped THEN
 			Configure := SetTrackObjName();
		END_IF
//----------------------------------------------------------------

	90: //Create some internal used variable
		THIS^.bNetworkHasTrackBranches := FALSE;
		THIS^.ipXpSystem.Tracks.ResetIterator();
		WHILE THIS^.ipXpSystem.Tracks.HasNextObject() DO
			IF __QUERYINTERFACE(THIS^.ipXpSystem.Tracks.GetNextObject(), ipEachTrack) AND_THEN (ipEachTrack.TracksAhead.Size > 1) THEN
				THIS^.bNetworkHasTrackBranches := TRUE;
				EXIT;
			END_IF
		END_WHILE
		THIS^.ipXpSystem.Tracks.RestoreIterator();
		
		

	100..CHALET_BaseComponents.GVL_Datatypes.cMaxUint: 
		// 100..MaxUint -> Invalide input
		Configure := E_FAIL;
		
	ELSE 
		//If an step is not defind/used return ok
		Configure := S_OK;
END_CASE


fbOptionalTrackUsedInLiveView.Update();
fbFeedback.Update();
END_METHOD

//This method is called when the system is disabled. Links are deleted as they may no longer be valid
METHOD Disassemble : HRESULT
VAR_INPUT
END_VAR
fbStationsAhead.Clear(); 
fbStationsBehinde.Clear(); 
fbListPathAhead.Clear(); 
fbListPathBehind.Clear(); 

Disassemble := S_OK;
END_METHOD

{attribute 'monitoring':='call'}
PROPERTY CtsEmptySpaceInQueue : UDINT
GET
//Handle UINT Overflow
IF THIS^.fbAssignedMovers.Size >= THIS^.nMoverQueueSize THEN
	CtsEmptySpaceInQueue := 0;
ELSE 
	CtsEmptySpaceInQueue := THIS^.nMoverQueueSize - THIS^.fbAssignedMovers.Size;
END_IF
END_GET
END_PROPERTY

{attribute 'monitoring':='call'}
PROPERTY CtsMoversInQueue : UDINT
GET
CtsMoversInQueue := THIS^.fbAssignedMovers.Size;
END_GET
END_PROPERTY

{attribute 'monitoring':='call'}
PROPERTY MoverAccAtExit : MC_LREAL //[mm/s² on Track] Every mover that leaves or passes the station gets this new acceleration as a target.
GET
MoverAccAtExit := THIS^.fMoverAccAtExit;
END_GET
SET
THIS^.fMoverAccAtExit := MoverAccAtExit;
END_SET
END_PROPERTY

{attribute 'monitoring':='call'}
PROPERTY MoverDecAtExit : MC_LREAL //[mm/s² on Track] Every mover that leaves or passes the station gets this new deceleration as a target.
GET
MoverDecAtExit := THIS^.fMoverDecAtExit;
END_GET
SET
THIS^.fMoverdecAtExit := MoverDecAtExit;
END_SET
END_PROPERTY

{attribute 'monitoring':='call'}
PROPERTY MoverQueueSize : UINT
GET
MoverQueueSize := THIS^.nMoverQueueSize;
END_GET
SET
THIS^.nMoverQueueSize := MoverQueueSize;
END_SET
END_PROPERTY

{attribute 'monitoring':='call'}
PROPERTY MoversInPlace : BOOL
GET
THIS^.Prepare();//Prepare time-critical information, if not already done


MoversInPlace := bMoversInPlace;
END_GET
END_PROPERTY

{attribute 'monitoring':='call'}
// Return a sorted list of movers in this zone. Index 0 is the mover in Front
PROPERTY MoversInQueue : REFERENCE TO ARRAY [0..(CHALET_BaseComponents.BaseParameterlist.MAX_OBJECTS-1)] OF I_XP_Mover_PLC
GET
MoversInQueue REF= THIS^.fbSortedListMoversInQueue.MoversInZone;
END_GET
END_PROPERTY

{attribute 'monitoring':='call'}
PROPERTY MoverVelocityAtExit : MC_LREAL //[mm/s on Track] Every mover that leaves or passes the station gets this new velocity as a target.
GET
MoverVelocityAtExit := THIS^.fMoverVeloAtExit;
END_GET
SET
THIS^.fMoverVeloAtExit := MoverVelocityAtExit;
END_SET
END_PROPERTY

METHOD PROTECTED OnMoverPasses : BOOL //This methode is called automaticly from the station and detect mover who is passing the station whitout be in queue.
VAR_INPUT
	ipMoverPasses : I_XP_Mover;
END_VAR
VAR
	ipThisStation : I_XP_Station := THIS^;
	
	//this raises an error 33155 "Target position is not reachable. There is no path available to the target position or target position is unreachable in general."
	bPreventMoveCmdToMoversCurrentPos : BOOL;
END_VAR
IF ipMoverPasses = 0 THEN
	RETURN;
END_IF


//Detect mover who is passing the station whitout be in queue. 
//Adjust to new Dynamics
IF NOT THIS^.bSuppressDynamicsChange AND XPlanarParameterlist.B_STATIONS_OVERRIDE_MOVER_DYN_CONSTRAINT THEN
	//Only if not in this queue
	IF ipMoverPasses.ParentStation <> ipThisStation  THEN
		ipMoverPasses.SetDynConstraint_Path(	V:= THIS^.fMoverVeloAtExit, 
												A:= THIS^.fMoverAccAtExit,
												D:= THIS^.fMoverDecAtExit,
												J:= MC_DEFAULT);
	END_IF
END_IF	



//Detect mover who is passing the station whitout be in queue. 
//Adjust to new Gap
IF NOT THIS^.bSuppressDynamicsChange THEN
	bPreventMoveCmdToMoversCurrentPos := (ipMoverPasses.PositionOnTrack = ipMoverPasses.LastCmdTargetPosition) AND (ipMoverPasses.CurrentTrack = ipMoverPasses.LastCmdTargetTrack);
	//Only if not in this queue
	IF ipMoverPasses.ParentStation <> ipThisStation AND NOT bPreventMoveCmdToMoversCurrentPos THEN
		ipMoverPasses.MoveOnTrack(ipTrack	:= ipMoverPasses.LastCmdTargetTrack,
								fPosition	:= ipMoverPasses.LastCmdTargetPosition, 
								fGap		:= THIS^.fMoverGapAtExit);
	END_IF
END_IF
END_METHOD

//The movers currently in this station must leave the station. 
//The movers actively search for a destination, but only leave if a new destination is available.
METHOD PushMoversOutOfStation : HRESULT
VAR_INPUT
END_VAR
THIS^.nCtsMoversMustLeaveThisStation := THIS^.CtsMoversInQueue;
END_METHOD

{attribute 'monitoring':='call'}
//prevent further movers from entering the station, 
//e.g. to prevent a collision. All movers that are already moving to reach this station will be stopped with a stop 
//and restarted with Ready True.
PROPERTY ReadyToRecvMovers : BOOL
GET
ReadyToRecvMovers := bReadyToRecvMovers;
END_GET
SET
VAR
	ipEachMover : I_XP_Mover;
END_VAR
(* zzz Todo braucht es das?
//Change to Not Ready:
IF (ReadyToRecvMovers = FALSE) AND (bReadyToRecvMovers <> ReadyToRecvMovers) THEN
	//halt all movers on the way
	fbAssignedMovers.ResetIterator();
	WHILE fbAssignedMovers.HasNextObject() DO
		IF ToXpMover(fbAssignedMovers.GetNextObject(),ipEachMover) THEN
			ipEachMover.Halt();	
		END_IF	
	END_WHILE
END_IF

//Change to Ready:
IF (ReadyToRecvMovers = TRUE) AND (bReadyToRecvMovers <> ReadyToRecvMovers) THEN
	//all movers that are on the way have probably been stopped before. when reactivated, the last move command is sent again.
	fbAssignedMovers.ResetIterator();
	WHILE fbAssignedMovers.HasNextObject() DO
		IF ToXpMover(fbAssignedMovers.GetNextObject(),ipEachMover) THEN
			ipEachMover.MoveOnTrack(ipTrack 	:= ipEachMover.LastCmdTargetTrack ,
									fPosition	:= ipEachMover.LastCmdTargetPosition,
									fGap		:= ipEachMover.LastCmdTargetGap);
		END_IF	
	END_WHILE
END_IF
*)
//Store new status
bReadyToRecvMovers := ReadyToRecvMovers;
END_SET
END_PROPERTY

METHOD SendMoversToStation : I_CH_Feedback //All movers in the station are sent to this destination
VAR_INPUT
	sTargetStation: STRING;//unique station name or group of stations
END_VAR
VAR
	nIdx : UDINT;
	ipXpMover : I_XP_Mover;
END_VAR
IF THIS^.fbFeedback.Error THEN
	//Error active/not ready
	THIS^.fbFeedback.LastCommandAccepted	:= FALSE;
	RETURN;
END_IF


//Invalide target
IF sTargetStation = '' THEN
	THIS^.fbFeedback.LastCommandAccepted	:= FALSE;
	RETURN;
END_IF


//Send all Queued movers away by changing the target station destination
THIS^.fbAssignedMovers.ResetIterator();
WHILE THIS^.fbAssignedMovers.HasNextObject() DO
	IF __QUERYINTERFACE(THIS^.fbAssignedMovers.GetNextObject(), ipXpMover) THEN
		
		ipXpMover.TargetStation := sTargetStation;	
		
	END_IF
END_WHILE
THIS^.fbAssignedMovers.RestoreIterator();


//A mover must leave the station immediately when the ‘SendMoversToStation’ method is called. The station is then available again.
//Otherwise, if no destination station is available, the mover waits in the station.
IF XPlanarParameterlist.B_MOVER_MUST_LEAVE_STATION_AT_SET_NEW_TARGED THEN
	//Mover must leave this station
	THIS^.PushMoversOutOfStation();
END_IF



SendMoversToStation := THIS^.fbFeedback;
END_METHOD

{attribute 'monitoring':='call'}
//Suppress to change the dynamic(Gap+velocity) of passing movers. This is usefull in startup
PROPERTY SuppressDynamicsChange : BOOL
GET
SuppressDynamicsChange := bSuppressDynamicsChange;
END_GET
SET
bSuppressDynamicsChange := SuppressDynamicsChange;
END_SET
END_PROPERTY

{attribute 'monitoring':='call'}
//Interface to CHALET system to which this object belongs
PROPERTY System : I_XP_System_PLC
GET
//get I_x_System_PLC interface from I_x_System_Registration
__QUERYINTERFACE(THIS^.ipXpSystem, System);
END_GET
END_PROPERTY

{attribute 'monitoring':='call'}
PROPERTY TargetGroupe : STRING
GET
TargetGroupe := THIS^.sTargetGroup;
END_GET
END_PROPERTY

{attribute 'monitoring':='call'}
//A time that is waited as soon as the mover is in the station (including the monitoring window) before “MoversInPlace” is set. e.g. used to stabilize the workpiece
PROPERTY TargetPosMonitoringTime : TIME
GET
TargetPosMonitoringTime := tTargetPosMonitoringTime;
END_GET
SET
tTargetPosMonitoringTime := TargetPosMonitoringTime;
END_SET
END_PROPERTY

{attribute 'monitoring':='call'}
//How many mm before the mover reaches the position is “MoversInPlace” set for the process. 
//This distance can also be set very large (e.g. 100mm) for moving past without stopping.
PROPERTY TargetPosWindow : LREAL
GET
TargetPosWindow := fTargetPosWindow;
END_GET
SET
fTargetPosWindow := TargetPosWindow;
END_SET
END_PROPERTY

{attribute 'monitoring':='call'}
PROPERTY ProcessSimulationActive : BOOL
GET
ProcessSimulationActive := THIS^.fSimulationProcessDuration > 0;
END_GET
END_PROPERTY

//If a valid time (>0seconds) is set and the configured destination station exists, then the movers will be sent away automatically after this time from now on.
METHOD SimulationStart : HRESULT
VAR_INPUT
	fProcessDuration 		: LREAL; //[s]
	sTargetStation	: STRING; //Group of the target station to automatic send after the duration
END_VAR
VAR
	ipStation	: I_CH_Object;
	ipXpSystemPlc : I_XP_System_PLC;
	bValideStation : BOOL;
END_VAR
bValideStation := __QUERYINTERFACE(THIS^.ipXpSystem,ipXpSystemPlc) AND ipXpSystemPlc <> 0 AND_THEN ipXpSystemPlc.CheckTargetExists(sTargetStation);

IF (fProcessDuration > 0) AND bValideStation THEN
	//Valide config
	THIS^.fSimulationProcessDuration 	:=	fProcessDuration;
	THIS^.sSimulationTargetStation 		:=	sTargetStation;
	SimulationStart := S_OK;
ELSE
	//Simulation disabled
	THIS^.fSimulationProcessDuration 	:=	0;
	THIS^.sSimulationTargetStation 		:=	'';
	SimulationStart := S_FALSE;
END_IF
END_METHOD

//If a valid time (>0seconds) is set and the configured destination station exists, then the movers will be sent away automatically after this time from now on.
METHOD SimulationStartEx : HRESULT
VAR_INPUT
	fProcessDuration 		: LREAL; //[s]
	ipStation				: I_XP_Station_PLC; //unique station to automatic send after the duration
END_VAR
VAR
	ipXpSystemPlc : I_XP_System_PLC;
	bValideStation : BOOL;
END_VAR
IF ipStation <> 0 THEN
	SimulationStartEx := THIS^.SimulationStart(fProcessDuration := fProcessDuration, sTargetStation := ipStation.LUID);

ELSE
	SimulationStartEx := S_FALSE;
END_IF
END_METHOD

METHOD SimulationStop : HRESULT
//Simulation disabled
THIS^.fSimulationProcessDuration 	:=	0;
THIS^.sSimulationTargetStation 		:=	'';
END_METHOD

METHOD PROTECTED UpdateSimulation : HRESULT
VAR_INST
	tonSimulationDelay : TON;
END_VAR
//Automatic send mover to next station in Simulation
//If a valid time (>0seconds) is set and the configured destination station exists, then the movers will be sent away automatically after this time from now on.
tonSimulationDelay.IN 	:= THIS^.ipXpSystem.Enabled AND THIS^.MoversInPlace AND THIS^.ProcessSimulationActive;
tonSimulationDelay.PT	:= LREAL_TO_TIME(THIS^.fSimulationProcessDuration*1000.0);
tonSimulationDelay();
IF tonSimulationDelay.Q THEN
	THIS^.SendMoversToStation(sTargetStation := THIS^.sSimulationTargetStation);
END_IF
END_METHOD

{attribute 'monitoring':='call'}
//Track on which the station is located
PROPERTY AccocietedTrack : I_XP_Track
GET
AccocietedTrack := THIS^.ipAccocietedTrack;
END_GET
END_PROPERTY

METHOD AddMoverToQueue : HRESULT
VAR_INPUT
	ipMover : I_XP_Mover;
END_VAR
//Get I_CH_Objekt of mover to put it in to a list.
IF ipMover <> 0 THEN
	//Add in List of Movers in this station
	THIS^.fbAssignedMovers.AddObject(ipMover);
	
	//Handover information in Mover
	ipMover.ParentStation := (THIS^);

	AddMoverToQueue := S_OK;
ELSE
	AddMoverToQueue := E_FAIL;;	
END_IF
END_METHOD

{attribute 'monitoring':='call'}
//List of movers managed by this station
PROPERTY AssignedMovers : I_CH_List
GET
AssignedMovers := THIS^.fbAssignedMovers;
END_GET
END_PROPERTY

{attribute 'monitoring':='call'}
(*[mm]
As soon as the mover is closer than this distance, the mover can be sent on to the next one if necessary.
This is the distance from the station to the end of the track or the shortest path to this station. Depending on which is closer. This is to ensure that the mover can no longer be overhauled.
This proberty can make the internal calculated distance smaller but not larger
Recalculated each disable/enable of the system*)
//Todo Increase shpuld also be possible
PROPERTY DecisionDistance : LREAL
GET
DecisionDistance := THIS^.fDecisionDistance;
END_GET
SET
THIS^.fDecisionDistance := MIN(THIS^.fDecisionDistance, ABS(DecisionDistance));
END_SET
END_PROPERTY

METHOD DeleteMoversQueue : HRESULT
VAR
	ipTempMover : I_XP_Mover;
END_VAR
//Not allowed in enabled state
IF THIS^.ipXPSystem.Enabled THEN
	DeleteMoversQueue := E_FAIL;
	RETURN;
END_IF


//Delete intormation in linked mover
THIS^.fbAssignedMovers.ResetIterator();
WHILE THIS^.fbAssignedMovers.HasNextObject() DO
	IF ToXPMover(THIS^.fbAssignedMovers.GetNextObject(),ipTempMover) THEN
		ipTempMover.ParentStation := 0;
	END_IF	
END_WHILE

//Clear list
fbAssignedMovers.Clear();

DeleteMoversQueue := S_OK;
END_METHOD

METHOD FB_exit : BOOL
VAR_INPUT
	bInCopyCode : BOOL; // if TRUE, the exit method is called for exiting an instance that is copied afterwards (online change).
END_VAR
VAR
	pFbPath : POINTER TO FB_XP_Path;
	ipObject : I_CH_Object;
END_VAR
// Not in an onlinechange - only in switch to configmode
IF NOT bInCopyCode THEN
	
	//Clear list, delete dynamic_creation path objects
	WHILE NOT THIS^.fbListPathAhead.IsEmpty DO
		ipObject := fbListPathAhead.GetRandomObject();
		fbListPathAhead.RemoveObject(ipObject);
		
		//Get pointer and delete
		IF __QUERYPOINTER(ipObject, pFbPath) THEN
			__DELETE(pFbPath);
		END_IF
	END_WHILE

END_IF
END_METHOD

METHOD FB_init : BOOL
VAR_INPUT
	bInitRetains : BOOL; // if TRUE, the retain variables are initialized (warm start / cold start)
	bInCopyCode : BOOL;  // if TRUE, the instance afterwards gets moved into the copy code (online change)
	
	ipSystem 			: I_CH_Object;
	ipAccocietedTrack 	: I_XP_Track;//track on which the station is located
	sUniqueName			: STRING;		//expl.:'Loading' unique identification for this station
	sTargetGroup		: STRING;	//to which group of stations does this station belong? e.g. several stations can belong to one 'Infeed' if this is implemented redundantly.
	nMoverQueueSize 	: UINT;
	xPos				: LREAL; 	
	yPos				: LREAL; 	
END_VAR
VAR 

END_VAR
//Do the following code once during start up and not during onlinechange
IF NOT bInCopyCode THEN 
	bErrorDuringFbInit := FALSE;
	
	(* Register to the Xplanar System
	   1. Test if the interface exists
	   2. Test if the object implements a "System for Mover" interface 
	*)
	IF ipSystem <> 0 AND_THEN __QUERYINTERFACE(ipSystem,THIS^.ipXpSystem) THEN
		THIS^.ipXpSystem.RegisterStation(THIS^);
	ELSE
		bErrorDuringFbInit := TRUE;
	END_IF

	THIS^.fbFeedback.ActiveCommand 		:= TO_STRING(THIS^.eActiveCommand);	
	
	// 0 = get closest track (in step configure)
	IF ipAccocietedTrack <> 0 THEN
		THIS^.ipAccocietedTrack := ipAccocietedTrack;
		bTrackIsSetInFbInit := TRUE;
	END_IF
	 
	
	//"" is maybe entered in an waiting or dynamic station and the name is not important
	IF sUniqueName <> '' THEN 
		THIS^.fbSourceInfo.sName := sUniqueName;
	ELSE
		sUniqueName := THIS^.fbSourceInfo.sName;
	END_IF

	
	//"" is maybe entered in an waiting or dynamic station and the name is not important
	IF sTargetGroup <> '' THEN 
		THIS^.sTargetGroup := sTargetGroup;
	ELSE
		THIS^.sTargetGroup := THIS^.fbSourceInfo.sName;
	END_IF

	
	THIS^.nMoverQueueSize 		:= nMoverQueueSize;
	THIS^.fbPositionPlanned.x 	:= xPos;
	THIS^.fbPositionPlanned.y 	:= yPos;


	THIS^.fbTrigger.FB_init(FALSE,FALSE, THIS^.ipXpSystem);

END_IF
END_METHOD

{attribute 'monitoring':='call'}
PROPERTY Feedback : I_CH_Feedback
GET
Feedback := THIS^.fbFeedback;
END_GET
END_PROPERTY

{attribute 'monitoring':='call'}
//Filter content, movers with one of these targets may not approach or drive over the station
PROPERTY Filter : STRING
GET
Filter := sFilter;
END_GET
SET
sFilter := Filter;
END_SET
END_PROPERTY

(*THIS METHOD uses the A* algorithm TO find the shortest route TO the destination in the network. Returns an INTERFACE with information about the destination found, such as station, path TO destination, path length.
If an interface=0 is returned, then no path can be found at the current time.*)
METHOD GetPathToTarget : I_PathAStarNode
VAR_INPUT
	sTargetStation : REFERENCE TO STRING; //unique station name or group of stations. EmptyString=Any
END_VAR
VAR	
	nDifZero : INT;	///zzz remove

	nIdx : UDINT;
	bCorrectLUID: BOOL;
	bCorrectGroupe : BOOL;
	bFilterBlockThisMover : BOOL;
	bStationIsBlocked : BOOL;
	bDummyStation : BOOL; //Station without movers only to change the dynamics of passing movers;
	bTargetFound : BOOL;
	bImTheAsker : BOOL; // Do not return this station as a target
	bStationCanNotBePassed : BOOL;
	
	
	ipActiveStationAStar : I_PathAStarNode;
	ipEmptyPathObj : I_PathAStarNode;
	ipEachPathAhead : I_XP_Path;
	ipPathFoundInOpenList : I_PathAStarNode;
	ipEachAStarNode : I_PathAStarNode;
	ipBesStationAStar : I_PathAStarNode;	
	ipThisStation : I_XP_Station := THIS^;
	
	fPathLength : LREAL;
END_VAR
VAR_INST
	fbLastFoundResult : FB_AStarNode;
END_VAR
VAR_STAT
	fbListNotUsedNodes : FB_CH_List; // Use GetNext() to allways get a not used one
	afbPathAStarNodes : ARRAY[0..(CHALET_BaseComponents.BaseParameterlist.MAX_OBJECTS-1)] OF FB_AStarNode;	
	fbListOpen : FB_CH_List; //To check
	fbListClosed : FB_CH_List; //Allready checked	
END_VAR
//only on first call, add nodes to list of not used objects
IF fbListNotUsedNodes.IsEmpty THEN
	FOR nIdx := 0 TO (CHALET_BaseComponents.BaseParameterlist.MAX_OBJECTS-1) DO
		fbListNotUsedNodes.AddObject(afbPathAStarNodes[nIdx]);
	END_FOR
END_IF

//Clear list
fbListOpen.Clear();
fbListClosed.Clear();

//Init objects in list
fbListNotUsedNodes.ResetIterator();
WHILE fbListNotUsedNodes.HasNextObject() DO
	IF __QUERYINTERFACE(fbListNotUsedNodes.GetNextObject(), ipEachAStarNode) THEN
		IF 	ipEachAStarNode.Station = 0 THEN
			EXIT;//Last used element found, abort
		END_IF
	
		ipEachAStarNode.Station := 0;
		ipEachAStarNode.RouteUsedToNode.Clear();
	END_IF
END_WHILE

//Reset last found result
fbLastFoundResult.Station := 0;
fbLastFoundResult.RouteUsedToNode.Clear();

// Reset once - Use GetNext() to allways get a not used one
fbListNotUsedNodes.ResetIterator();

//This is the start of the search operation. Add this station
__QUERYINTERFACE(fbListNotUsedNodes.GetNextObject(), ipEmptyPathObj);
ipEmptyPathObj.Station := (THIS^);
fbListOpen.AddObject(ipEmptyPathObj);

WHILE NOT fbListOpen.IsEmpty DO
	//Get objet from list with smallest distanse to start-station

	__QUERYINTERFACE(fbListOpen.GetObjectWithLowestNumber(), ipActiveStationAStar);
	//Move objet from open to closed list
	fbListOpen.RemoveObject(ipActiveStationAStar);
	fbListClosed.AddObject(ipActiveStationAStar);
	
	IF ipBesStationAStar <> 0 AND_THEN ipActiveStationAStar.PathLength > ipBesStationAStar.PathLength THEN
		// if a valid station is allreadyx known, skip all station who allready have a larger distance
		CONTINUE;
	END_IF
	
	bImTheAsker := ipActiveStationAStar.Station = ipThisStation;
	bCorrectLUID := (ipActiveStationAStar.Station.LUID = sTargetStation);
 	bCorrectGroupe := (ipActiveStationAStar.Station.TargetGroupe = sTargetStation) OR (sTargetStation =  XPlanarParameterlist.S_ANY_STATION_NAME);
	bDummyStation := (ipActiveStationAStar.Station.MoverQueueSize = 0);//Station without movers only to change the dynamics of passing movers;
	bFilterBlockThisMover := (ipActiveStationAStar.Station.Filter <>  XPlanarParameterlist.S_ANY_STATION_NAME) AND (ipActiveStationAStar.Station.Filter <> sTargetStation) AND NOT bCorrectLUID; // Correct LUID is stronger than filter
	bStationIsBlocked := (ipActiveStationAStar.Station.CtsEmptySpaceInQueue <= 0 AND NOT bDummyStation) OR NOT ipActiveStationAStar.Station.ReadyToRecvMovers;
	bStationCanNotBePassed := ipActiveStationAStar.Station.CtsMoversInQueue > 0 AND NOT bImTheAsker ;
	
	IF (bFilterBlockThisMover OR bStationIsBlocked) AND NOT bImTheAsker THEN
		//Skip
		CONTINUE;
	END_IF
	
	
	IF (bCorrectLUID OR bCorrectGroupe) AND NOT bImTheAsker AND NOT bDummyStation THEN
		//FOUND! - check if way is shorter
		IF ipBesStationAStar=0 OR_ELSE  ipActiveStationAStar.PathLength <= ipBesStationAStar.PathLength THEN
			//shorter - store
			ipBesStationAStar := ipActiveStationAStar;
		END_IF
		
	ELSIF NOT bStationCanNotBePassed THEN		
		// If the destination has not yet been found, set the successor nodes of the current node to the open list
		ipActiveStationAStar.Station.PathsAhead.ResetIterator();
		WHILE ipActiveStationAStar.Station.PathsAhead.HasNextObject() DO
			__QUERYINTERFACE(ipActiveStationAStar.Station.PathsAhead.GetNextObject(), ipEachPathAhead); 
			
			IF fbListClosed.LUIDInList(ipEachPathAhead.StationDestination.LUID) THEN
				// if the successor node is already on the closed list - do nothing, repeate WHILE loop
				CONTINUE;
			END_IF
			
			//Calculate distance to start oh the new found station
			fPathLength := ipActiveStationAStar.PathLength + ipEachPathAhead.Length;
		
			//Check if this station is allready existin in open list - compare if this one is shorter
			IF __QUERYINTERFACE( fbListOpen.FindLUID(ipEachPathAhead.StationDestination.LUID), ipPathFoundInOpenList)  THEN
				IF ipPathFoundInOpenList.PathLength <= fPathLength  THEN
					//object in open list is shorter - do nothing, repeate WHILE loop
					CONTINUE;
				ELSE
					//new object is shorter - remove old object in open lsit
					fbListOpen.RemoveObject(ipPathFoundInOpenList);
				END_IF
			END_IF			
			
			
			//Add this path ahead to open list - set new length
			__QUERYINTERFACE(fbListNotUsedNodes.GetNextObject(), ipEmptyPathObj);
			ipEmptyPathObj.Station := ipEachPathAhead.StationDestination;
			ipEmptyPathObj.RouteUsedToNode.Duplicate(ipActiveStationAStar.RouteUsedToNode);
			ipEmptyPathObj.RouteUsedToNode.AddObject(ipEachPathAhead);
			fbListOpen.AddObject(ipEmptyPathObj);

		END_WHILE
		ipActiveStationAStar.Station.PathsAhead.RestoreIterator();

	END_IF

END_WHILE


//Return station or nothing
IF ipBesStationAStar = 0 THEN
	GetPathToTarget := 0;
ELSE
	//store list in an instance
	fbLastFoundResult.Station := ipBesStationAStar.Station;
	fbLastFoundResult.RouteUsedToNode.Duplicate(ipBesStationAStar.RouteUsedToNode);
	GetPathToTarget := fbLastFoundResult;
END_IF
END_METHOD

METHOD Initialize : HRESULT
VAR
	ipEachStationAhead : I_XP_Station;
	nIdx : UDINT;
END_VAR
VAR_INST
	//This error cannot be reset. Requires a reset cold
	{attribute 'hide'}	
	fbInitError : FB_TcAlarm;
	{attribute 'hide'}	
	fbMissingInterfaceAlarm : FB_TcAlarm;
END_VAR
//Check Error during FB_Init
IF THIS^.bErrorDuringFbInit THEN
	IF NOT fbInitError.bRaised THEN 
		//This error cannot be reset. Requires a reset cold
		fbInitError.CreateEx(stEventEntry:=TC_EVENTS.CHALET_Base_Events.ErrorFBinit, ipSourceInfo := THIS^.fbSourceInfo, bWithConfirmation := FALSE);
		fbInitError.Raise(0);
	END_IF
	Initialize:= E_FAIL;
	THIS^.fbFeedback.HR := Initialize;
	RETURN;
END_IF	

//Interface to System is missing
IF THIS^.ipXpSystem = 0 THEN
	IF NOT fbMissingInterfaceAlarm.bRaised THEN 
		//This error cannot be reset. Requires a reset cold
		fbMissingInterfaceAlarm.CreateEx(stEventEntry:=TC_EVENTS.CHALET_Base_Events.ErrorFBinit, ipSourceInfo := THIS^.fbSourceInfo, bWithConfirmation := FALSE);
		fbMissingInterfaceAlarm.Raise(0);
	END_IF
	Initialize := E_FAIL;
	THIS^.fbFeedback.HR := Initialize;
	RETURN;
END_IF


IF NOT THIS^.bInitDone THEN
	//Busy
	Initialize:= S_PENDING;
	
	//Clean up
	THIS^.DeleteMoversQueue();


	bInitDone := TRUE;
ELSE
	//Done
	Initialize:= S_OK;
END_IF


THIS^.eActiveCommand 				:= CHALET_NC.E_NcAxisCommands.Initialize;
THIS^.fbFeedback.ActiveCommand 		:= TO_STRING(THIS^.eActiveCommand);	
THIS^.fbFeedback.LastCommandAccepted:= TRUE;	
//Set done or keep in busy state	
THIS^.fbFeedback.HR := Initialize;
END_METHOD

{attribute 'monitoring':='call'}
//[mm] Every mover that leaves or passes the station gets this new gap as a target.
PROPERTY MoverGapAtExit : LREAL
GET
MoverGapAtExit := fMoverGapAtExit;
END_GET
SET
IF MoverGapAtExit < XPlanarParameterlist.F_MOVER_MINIMUM_GAP_ON_TRACK THEN
	MoverGapAtExit := XPlanarParameterlist.F_MOVER_MINIMUM_GAP_ON_TRACK;
END_IF

fMoverGapAtExit := MoverGapAtExit;
END_SET
END_PROPERTY

{attribute 'monitoring':='call'}
//Unique object ID
PROPERTY OID : OTCID
GET
OID := THIS^.fbOptionalTrackUsedInLiveView.MCTOPLC_STD.TrackOID;
END_GET
END_PROPERTY

{attribute 'monitoring':='call'}
//List of paths that lead to stations before this station
PROPERTY PathsAhead : I_CH_List
GET
PathsAhead := THIS^.fbListPathAhead;
END_GET
END_PROPERTY

{attribute 'monitoring':='call'}
//List of paths that lead to stations behind this station
PROPERTY PathsBehinde : I_CH_List
GET
PathsBehinde := THIS^.fbListPathBehind;
END_GET
END_PROPERTY

{attribute 'monitoring':='call'}
//[mm] from the beginning of the assigned track
PROPERTY PositionOnTrack : LREAL
GET
PositionOnTrack := THIS^.fPositionOnTrack;
END_GET
END_PROPERTY

{attribute 'monitoring':='call'}
//Position on the assigned track
PROPERTY PositionOnTrackXY : REFERENCE TO PositionXY
GET
PositionOnTrackXY REF= THIS^.fbPositionOnTrackXY;
END_GET
END_PROPERTY

{attribute 'monitoring':='call'}
//Position on the assigned track
PROPERTY PositionOnTrackXYZABC : REFERENCE TO MoverVector
GET
VAR_INST
	{attribute 'hide'}
	stPosOnTrack : MoverVector;
END_VAR
stPosOnTrack.x := fbPositionOnTrackXY.x;
stPosOnTrack.y := fbPositionOnTrackXY.y;
stPosOnTrack.z := 0;
stPosOnTrack.a := 0;
stPosOnTrack.b := 0;
stPosOnTrack.c := 0;

PositionOnTrackXYZABC REF= stPosOnTrack;
END_GET
END_PROPERTY

{attribute 'monitoring':='call'}
//Planned position, not necessarily on the track. Only changeable when the system is disabled
PROPERTY PositionXY : REFERENCE TO  PositionXY
GET
PositionXY REF= THIS^.fbPositionPlanned;
END_GET
END_PROPERTY

(* 
	Use this Methode to calculate time sensitive date once each cycle. Example: read analog input and convert before do get Signal propertie
*)
METHOD PROTECTED Prepare : HRESULT
VAR_INST
	{attribute 'hide'}	
	nLastUpdatedCycleCount : UDINT;
END_VAR

VAR
	nLoopIndex : UINT;
	fExpectedDistanceToParent : LREAL;
	nCycleTime_ms : UDINT;
	bMoverInQueue : BOOL;
	bTempMoverInPosition : BOOL;
	bTempMoverVeloZero : BOOL;
	bTempMoverInMonitoringTime : BOOL;
	bTempMoverThisStationAsTarget : BOOL;
END_VAR
VAR_INST
	{attribute 'hide'}
	nCycleCountInPos : UDINT;
END_VAR
//Check if this Cycle the dates are allready prepared. This is important for time sensitive informations.
IF nLastUpdatedCycleCount <> TwinCAT_SystemInfoVarList._TaskInfo[THIS^.TaskIndex].CycleCount THEN
	nLastUpdatedCycleCount := TwinCAT_SystemInfoVarList._TaskInfo[THIS^.TaskIndex].CycleCount ;


	(* Check if mover is in place. Time and Position window *)
	//If queuesize is zero, mover is never in place.
	IF nMoverQueueSize = 0 OR THIS^.ipAccocietedTrack = 0 OR NOT ipXpSystem.Enabled THEN
		THIS^.bMoversInPlace := FALSE;
		nCycleCountInPos := 0;
	ELSE
		//Get this task cycle Count and time 
		nCycleTime_ms := TwinCAT_SystemInfoVarList._TaskInfo[THIS^.nTaskIndex].CycleTime(*100ns*) / 10_000 ;
		
		bTempMoverInPosition := TRUE; bTempMoverVeloZero := TRUE; bTempMoverThisStationAsTarget := TRUE;
		fExpectedDistanceToParent := 0;
		FOR nLoopIndex := 0 TO (THIS^.nMoverQueueSize-1) DO
			IF THIS^.fbSortedListMoversInQueue.MoversInZone[nLoopIndex] <> 0 THEN
				//Check position and Gap - 1 mover do not have a gap
				IF nLoopIndex <> 0 THEN
					fExpectedDistanceToParent := fExpectedDistanceToParent + THIS^.fbSortedListMoversInQueue.MoversInZone[nLoopIndex].LastCmdTargetGap;
				END_IF
				bMoverInQueue		:= TRUE;
				bTempMoverInPosition := bTempMoverInPosition AND (ABS(THIS^.fbSortedListMoversInQueue.MoversInZone[nLoopIndex].DistToParentStation - fExpectedDistanceToParent) <= fTargetPosWindow );
				bTempMoverVeloZero := bTempMoverVeloZero AND (THIS^.fbSortedListMoversInQueue.MoversInZone[nLoopIndex].PlanarMover.MCTOPLC.SETONTRACK.SetVelo = 0.0);
				bTempMoverThisStationAsTarget := bTempMoverThisStationAsTarget AND ((THIS^.fbSortedListMoversInQueue.MoversInZone[nLoopIndex].TargetStation = THIS^.TargetGroupe) OR (THIS^.fbSortedListMoversInQueue.MoversInZone[nLoopIndex].TargetStation = THIS^.LUID));
			ELSE
				//Missing mover in queue
				bMoverInQueue := FALSE;
				EXIT;
			END_IF
		END_FOR
			
		//start time if mover position is ok
		IF bTempMoverInPosition  THEN
			nCycleCountInPos := nCycleCountInPos + 1;
		ELSE
			nCycleCountInPos := 0;
		END_IF
		
		bTempMoverInMonitoringTime := (UDINT_TO_TIME(nCycleCountInPos * nCycleTime_ms) >= tTargetPosMonitoringTime);
				
		THIS^.bMoversInPlace := bMoverInQueue AND bTempMoverInPosition AND bTempMoverInMonitoringTime AND bTempMoverThisStationAsTarget;// AND bTempMoverVeloZero;
	END_IF
	
	
END_IF
END_METHOD

{attribute 'monitoring':='call'}
//List of stations before this station
PROPERTY StationsAhead : I_CH_List
GET
StationsAhead := THIS^.fbStationsAhead;
END_GET
END_PROPERTY

{attribute 'monitoring':='call'}
//List of stations behinde this station
PROPERTY StationsBehinde : I_CH_List
GET
StationsBehinde := THIS^.fbStationsBehinde;
END_GET
END_PROPERTY

METHOD Update : HRESULT
VAR
	nIdx : UDINT;
	bStationIsBlocked : BOOL;
	ipThisStation : I_XP_Station := THIS^;
END_VAR
//Force to do init befor call update
IF NOT bInitDone THEN
	THIS^.Initialize();
	RETURN;
END_IF

THIS^.Prepare();//Prepare time-critical information, if not already done


// ********************** Set feedback depending on active command *******************************
CASE THIS^.eActiveCommand OF

	E_NcAxisCommands.Initialize:
		fbFeedback.Busy 			:= NOT THIS^.bInitDone;
		fbFeedback.Done 			:= THIS^.bInitDone;
		fbFeedback.ErrorId 			:= 0;
		                        	

	ELSE//External command in subclass
		;
END_CASE


// **********************  Stop to execute commands on .done or .error ***************************
IF fbFeedback.Done OR THIS^.fbFeedback.Error THEN
	eActiveCommand 				:= E_NcAxisCommands.None;
END_IF



// **********************  OnMoverPasses ***************************
// Detect mover who is passing the station and call method for easier overwriting
IF fbTrigger.MoverDetected AND (fbTrigger.MoverAtTrigger <> 0) AND_THEN (fbTrigger.MoverAtTrigger.ParentStation <> ipThisStation) THEN
	THIS^.OnMoverPasses(fbTrigger.MoverAtTrigger);
END_IF


// **********************  If enabled start station logic ***************************
IF THIS^.ipXpSystem.Enabled THEN
	
	// Process Simulation. 	
	// All functionality packed into one method for easier overwriting
	THIS^.UpdateSimulation();
	
		
	// Interaction with the movers. Sending on to the next station. 
	// All functionality packed into one method for easier overwriting
	THIS^.UpdateMoverInteraction();
	
	
	//Check for errors
	(*The station is blocked. 
	The first mover in the row is correctly positioned in the station. 
	The queue has a size of >1, but now the n+1 mover does not have this station as its destination. 
	However, it cannot overtake. The station never gives the process a ready signal.*)
	IF THIS^.MoverQueueSize > 1 AND THIS^.MoversInQueue[0] <> 0 AND_THEN (THIS^.MoversInQueue[0].TargetStation = THIS^.TargetGroupe OR THIS^.MoversInQueue[0].TargetStation = THIS^.LUID) THEN
		FOR nIdx := 1 TO (CHALET_BaseComponents.BaseParameterlist.MAX_OBJECTS-1) DO
			//Search for Mover with a direrent target
			IF THIS^.MoversInQueue[nIdx] <> 0 AND_THEN NOT(THIS^.MoversInQueue[nIdx].TargetStation = THIS^.TargetGroupe OR THIS^.MoversInQueue[nIdx].TargetStation = THIS^.LUID) THEN
				//Error
				bStationIsBlocked := TRUE;
				IF NOT fbAlarmStationIsBlocked.bRaised THEN
					//Station is blocked. Mover {0} has {1} as target position but cannot overtake
					fbAlarmStationIsBlocked.CreateEx(TC_Events.CHALET_XPlanar_Events.StationIsBlocked,0,THIS^.fbSourceInfo);
					fbAlarmStationIsBlocked.ipArguments.AddStringByValue(THIS^.MoversInQueue[nIdx].LUID).AddStringByValue(THIS^.MoversInQueue[nIdx].TargetStation);
					fbAlarmStationIsBlocked.Raise(0);
					EXIT;					
				END_IF
			END_IF
		END_FOR
	END_IF
	IF NOT bStationIsBlocked AND fbAlarmStationIsBlocked.bRaised THEN
		fbAlarmStationIsBlocked.Clear(0,0);
	END_IF
	
	
END_IF



// **********************  If disabled clear some bits ***************************
IF NOT THIS^.ipXpSystem.Enabled THEN
	fbAlarmStationIsBlocked.Clear(0,0);
END_IF

Update := S_OK;
END_METHOD

METHOD PROTECTED UpdateMoverInteraction : HRESULT
VAR
	ipFirstMoverInQueue: I_XP_Mover;
	sTargetStation : STRING;
	bMoverValideToSendAway : BOOL;
	bInReachForNewCmd : BOOL;
	bThisStationAsParent : BOOL;
	bFilterDoesNotAllowThisMover : BOOL;
	bThisStationAsTarget : BOOL;
	bMoverIsNotOnAWaitingStation : BOOL;
	bStationInBlockedTryToSolve : BOOL; //Send 1. Mover away ignore that already in correct station
	bMoverMustLeaveTheStation : BOOL; //Set from external
	bSearchNewDestination : BOOL;
	bStationCanBeReachedWhitoutBranch : BOOL;
	bStationIsOverfilled : BOOL;

	ipStationAhead : I_XP_Station;
	ipPathFoundAStarValide : I_PathAStarNode;
	ipPathFoundAStarAnyStation : I_PathAStarNode;
	ipRouteUsed : I_XP_Path;
	
	fbListOf : FB_AStarNode;
	
	
	ipThisStation : I_XP_Station := THIS^;
	ipPath : I_XP_Path;
	ipRoute : I_CH_List;
	ipMover : I_XP_Mover;
	fDistToThisStation : LREAL;
	bValideStationToStartMove : BOOL;
	bValideInterface, bMoverOnSameTrack, bInDecisionDistance : BOOL;
END_VAR
//Get first mover in this station
IF __QUERYINTERFACE(THIS^.MoversInQueue[0],ipFirstMoverInQueue) THEN

	//Get a few helpful variables
	sTargetStation := ipFirstMoverInQueue.TargetStation;
	bThisStationAsTarget := (sTargetStation = THIS^.TargetGroupe) OR (sTargetStation = THIS^.LUID); 
	bThisStationAsParent := ipFirstMoverInQueue.ParentStation.LUID = THIS^.LUID;
	bMoverIsNotOnAWaitingStation := NOT(bThisStationAsParent AND NOT bThisStationAsTarget AND (THIS^.MoverQueueSize > 0));
	bInReachForNewCmd	:= (ipFirstMoverInQueue.DistToParentStation <= THIS^.fDecisionDistance);	
	bStationInBlockedTryToSolve  := THIS^.fbAlarmStationIsBlocked.bRaised;//Send 1. Mover away ignore that already in correct station
	bFilterDoesNotAllowThisMover := (THIS^.Filter <> XPlanarParameterlist.S_ANY_STATION_NAME) AND (THIS^.Filter <> sTargetStation);
	bMoverMustLeaveTheStation := THIS^.nCtsMoversMustLeaveThisStation > 0;
	bStationIsOverfilled  := THIS^.CtsMoversInQueue > THIS^.nMoverQueueSize;
	
	
	//Decide what happens to the mover
	bSearchNewDestination := bInReachForNewCmd AND bThisStationAsParent AND (NOT bThisStationAsTarget OR bMoverMustLeaveTheStation OR bStationInBlockedTryToSolve OR bStationIsOverfilled);
	IF bSearchNewDestination THEN

	
		//1. Prio - Get a direct path to target - Only if specific
		IF sTargetStation <> XPlanarParameterlist.S_ANY_STATION_NAME THEN
			ipPathFoundAStarValide := GetPathToTarget(sTargetStation := sTargetStation);
		END_IF
	
		
		
		//If path to target is not valide, calculate once a path to any station
		IF ipPathFoundAStarValide = 0 THEN
			ipPathFoundAStarAnyStation := THIS^.GetPathToTarget(sTargetStation := XPlanarParameterlist.S_ANY_STATION_NAME);
		END_IF
		
		
		//2. Prio If the next possible station is on this track, without having to pass a switch, then go to this new station
		// The mover should be pushed as far forward as possible to avoid blocking the track
		IF  ipPathFoundAStarValide = 0 AND ipPathFoundAStarAnyStation <> 0  AND (THIS^.PathsAhead.Size = 1) AND THIS^.bNetworkHasTrackBranches THEN
			//
			ipPathFoundAStarAnyStation.RouteUsedToNode.ResetIterator();
			bStationCanBeReachedWhitoutBranch := TRUE;
			WHILE (ipPathFoundAStarAnyStation.RouteUsedToNode.HasNextObject() AND bStationCanBeReachedWhitoutBranch) DO
				IF __QUERYINTERFACE(ipPathFoundAStarAnyStation.RouteUsedToNode.GetNextObject(), ipRouteUsed) THEN
					bStationCanBeReachedWhitoutBranch := (ipRouteUsed.StationDestination.PathsAhead.Size = 1) OR (ipRouteUsed.StationDestination = ipPathFoundAStarAnyStation.Station); //Ignore if destination station have more than 1 paths ahead
				END_IF
			END_WHILE	
			ipPathFoundAStarAnyStation.RouteUsedToNode.RestoreIterator();
			IF bStationCanBeReachedWhitoutBranch THEN
				ipPathFoundAStarValide := ipPathFoundAStarAnyStation;
			END_IF
		END_IF
	
		
		//3. Prio - Send the mover to any station. (most time waitingstation)
		// - closest waitingstation to this station, if not allready on a waiting station
		// - if filter was maybe changed or the mover is not allowed in this station
		IF  ipPathFoundAStarValide = 0 AND ipPathFoundAStarAnyStation <> 0 AND (bMoverIsNotOnAWaitingStation OR bFilterDoesNotAllowThisMover OR bMoverMustLeaveTheStation OR bStationIsOverfilled) THEN
			ipPathFoundAStarValide := ipPathFoundAStarAnyStation;
		END_IF
	END_IF
	
	
	//Write new paths and parent-station to mover
	IF ipPathFoundAStarValide <> 0 THEN 
		//Handover list of paths to mover
		ipFirstMoverInQueue.SetRouteToParent(ipPathFoundAStarValide.RouteUsedToNode);
	
		//Unregister from this station and register with a new parrent station
		THIS^.fbAssignedMovers.RemoveObject(ipFirstMoverInQueue);
		ipPathFoundAStarValide.Station.AddMoverToQueue(ipFirstMoverInQueue);	
		
		//Mover is now leaving the station
		IF THIS^.nCtsMoversMustLeaveThisStation > 0 THEN
			THIS^.nCtsMoversMustLeaveThisStation := THIS^.nCtsMoversMustLeaveThisStation - 1;
		END_IF
		
	END_IF     
END_IF



//---------------------------------------------------------------
//- Update movers not in this queue unsig the route informations
//---------------------------------------------------------------

//The movers have a list of waypoints that they have to travel to on the way to the destination station. 
//It is checked whether this station is one of these waypoints
// - if yes, send the mover to the next waypoint and remove this stop from the list
//Do not wait until mover is at station possition, use fDecisionDistance
ipXpSystem.MoversPresent.ResetIterator();
WHILE ipXpSystem.MoversPresent.HasNextObject() DO
	IF __QUERYINTERFACE(ipXpSystem.MoversPresent.GetNextObject(),ipMover) THEN
		ipRoute := ipMover.RouteRemaining;
		bValideInterface 	:= ipRoute <> 0;
		bMoverOnSameTrack 	:= ipMover.CurrentTrack = ipThisStation.AccocietedTrack;
		fDistToThisStation  := F_GetDistToPosModulo(fTargetPosition := ipThisStation.PositionOnTrack, fActualPosition := (ipMover.PositionOnTrack-1.0), fModulo :=ipThisStation.AccocietedTrack.Length); 
		bInDecisionDistance := (fDistToThisStation <= THIS^.fDecisionDistance);
	ELSE 
		CONTINUE;
	END_IF		
	
	IF bValideInterface AND bMoverOnSameTrack AND bInDecisionDistance THEN
		ipRoute.ResetIterator();
		WHILE ipRoute.HasNextObject() DO
			IF __QUERYINTERFACE(ipRoute.GetNextObject(), ipPath) AND_THEN ipPath.StationStart = ipThisStation THEN
				//Remove this path from route and send to path desination
				ipMover.RouteSegmentDone(ipPath);
				
				//This is normal behavior if not a parent station. 
				//The mover is ~fDecisionDeistance away from the station and is given a new target position to travel further without reducing speed
				IF (fDistToThisStation > 1.0) THEN
					ipMover.MoveOnTrackToStation(ipStation := ipPath.StationDestination,
												fGap:= ipMover.LastCmdTargetGap);
				END_IF	
				 
				 
				//If the mover is very close to the transition, the next settings are already used here
				//This is the case if the mover was in a station for an interaction.
				IF (fDistToThisStation <= 1.0) THEN
					//Set new dynamic. Be careful when reducing the deceleration so that the mover can still stop in real time
					IF XPlanarParameterlist.B_STATIONS_OVERRIDE_MOVER_DYN_CONSTRAINT THEN
						ipMover.SetDynConstraint_Path(	V:= THIS^.fMoverVeloAtExit, 
														A:= THIS^.fMoverAccAtExit,
														D:= THIS^.fMoverDecAtExit,
														J:= MC_DEFAULT);
					END_IF
					ipMover.MoveOnTrackToStation(	ipStation := ipPath.StationDestination,
													fGap := THIS^.fMoverGapAtExit);	
				END_IF	
			END_IF
		END_WHILE
		ipRoute.RestoreIterator();
	END_IF		
END_WHILE
ipXpSystem.MoversPresent.RestoreIterator();
END_METHOD

END_FUNCTION_BLOCK

// COMPONENTs/System/FB_XP_System
{attribute 'no_explicit_call' := 'Do not call the body - Stick to OOP'}
(* XPlanar System - 1 per associated XPlanar 
	The system is the container and organizer for all subsequent XPlanar objects. All objects are registered with this system*)
FUNCTION_BLOCK FB_XP_System EXTENDS FB_CH_Object IMPLEMENTS I_XP_System_Registration, I_XP_System_PLC
VAR	
	{attribute 'hide'}
	bInitDone : BOOL;
	{attribute 'hide'}
	bErrorDuringFbInit : BOOL; // Not possible to reset
	{attribute 'hide'}                   	
	eActiveCommand 		: CHALET_Nc.E_NcAxisCommands := CHALET_Nc.E_NcAxisCommands.None;
	{attribute 'hide'}
    fbMoversPresent     : FB_CH_List;
	{attribute 'hide'}
    fbMoversNotPresent 	: FB_CH_List;
	{attribute 'hide'}
	fbListAllMovers 	: FB_CH_List;
	{attribute 'hide'}	
    fbTracks    		: FB_CH_List;
	{attribute 'hide'}	
	fbStationsAll 	 : FB_CH_List;//List of all station objects that exist in this project
	{attribute 'hide'}	
	fbStationsUsed 	 : FB_CH_List;//List of all station objects that are considered for path planning in the currently running system
	{attribute 'hide'}	
	fbTriggers 	 : FB_CH_List;
	{attribute 'hide'}	
	fbZones 	 : FB_CH_List;
	{attribute 'hide'}	
	fbPaths 	 : FB_CH_List;
	{attribute 'hide'}	
    ipGroup       : I_XP_Group;
	{attribute 'hide'}	
    ipEnvironment : I_XP_Environment;
	{attribute 'hide'}
    nSeqEnabling  : UINT;
	{attribute 'hide'}
	nSeqJoiningTrack : UINT;
	{attribute 'hide'}
	nSeqJoiningStation : UINT;
	{attribute 'hide'}	
    nSeqDisabling  : UINT := SEQ_DONE;
	{attribute 'hide'}
	fbFeedback : FB_CH_Feedback(ipSourceInfo := fbSourceInfo);	
END_VAR
VAR CONSTANT
	{attribute 'hide'}
	SEQ_DONE : UINT := 999;
END_VAR

METHOD AddMoverToSystem : HRESULT
VAR_INPUT
	ipMover : I_XP_Mover;
	xPos, yPos : LREAL;
END_VAR
VAR
	stParameter : EnterOrLeaveMovementAreaParameters;
END_VAR
IF ipMover <> 0 THEN
	THIS^.fbMoversNotPresent.RemoveObject(ipMover);
	
	//Add if not already in list
	IF NOT THIS^.fbMoversPresent.ObjectInList(ipMover) THEN
		THIS^.fbMoversPresent.AddObject(ipMover);
	END_IF
	
	//todo
//	stParameter.
//	ipMover.TcIoXPlanarMover.SetMovementArea(stParameter);
END_IF
END_METHOD

METHOD RemoveMoverFromSystem : HRESULT
VAR_INPUT
	ipMover : I_XP_Mover;
END_VAR

IF ipMover <> 0 THEN
	THIS^.fbMoversPresent.RemoveObject(ipMover);
	
	ipMover.Disassemble();
	
	
	//Add if not already in list
	IF NOT THIS^.fbMoversNotPresent.ObjectInList(ipMover) THEN
		THIS^.fbMoversNotPresent.AddObject(ipMover);
	END_IF
END_IF
END_METHOD

METHOD PROTECTED JoiningStation : HRESULT
VAR
	hr : HRESULT;
	ipEachMover : I_XP_Mover;
	ipEachMoverPlc : I_XP_Mover_PLC;
	ipEachMoverInStation : I_XP_Mover;
	ipEachStation : I_XP_Station;
	ipFirstStation : I_XP_Station;
	ipParentStation : I_XP_Station;
	ipTempMoverPlc : I_XP_Mover_PLC;

	//during move on track
	fVelo	: Tc3_Mc3Definitions.MC_LREAL := Tc3_Mc3Definitions.MC_DEFAULT; 
	fAccDec	: Tc3_Mc3Definitions.MC_LREAL := Tc3_Mc3Definitions.MC_DEFAULT;
	bError : BOOL;
	bFound : BOOL;
	bMoverAtCmdPos : BOOL;
	refPosition : REFERENCE TO MoverVector;
	fCalcualtedGapAtMoverPosition : LREAL;

	ipClosestStation : I_XP_Station;
	fDistToStation : LREAL := CHALET_BaseComponents.GVL_Datatypes.cMaxLreal;
END_VAR
VAR_INST
	bResetMovers : BOOL;	

	{attribute 'hide'}	
	fbDelayJoiningStation : TON;
END_VAR
CASE nSeqJoiningStation OF

	0: //Init
		fbDelayJoiningStation.IN := FALSE;
		
		IF fbStationsUsed.IsEmpty THEN
			nSeqJoiningStation := SEQ_DONE;
		ELSE
			nSeqJoiningStation := 10;
		END_IF
	


	
		
	10:	// For each Mover, Clear planed route to target. After enabling the tracks may have change and are not longer existing.
		THIS^.fbMoversPresent.ResetIterator();
		WHILE THIS^.fbMoversPresent.HasNextObject() DO
			IF __QUERYINTERFACE(THIS^.fbMoversPresent.GetNextObject(), ipEachMover) THEN
				//clear route
				ipEachMover.SetRouteToParent(0);
			END_IF
		END_WHILE
		THIS^.fbMoversPresent.RestoreIterator();
		
		//Empty Mover queue in station
		THIS^.fbStationsUsed.ResetIterator();
		WHILE THIS^.fbStationsUsed.HasNextObject() DO
			IF __QUERYINTERFACE(THIS^.fbStationsUsed.GetNextObject(), ipEachStation) THEN
				ipEachStation.DeleteMoversQueue(); // This is also reset the parent of each mover
			END_IF
		END_WHILE
		THIS^.fbStationsUsed.RestoreIterator();
		
		nSeqJoiningStation := 20;
	
	


	
		
	20: (*Check whether the last set station parent (station responsible for continuing to send the mover) is still valid. This is not the case if, for example:
		- Mover was manually moved to a new position
		- Track layout has changed
		- Position of the station has changed - No longer exists	*)
		THIS^.fbMoversPresent.ResetIterator();
		WHILE THIS^.fbMoversPresent.HasNextObject() DO
			IF __QUERYINTERFACE(THIS^.fbMoversPresent.GetNextObject(), ipEachMover) THEN
				//Prio 1: If the station ahead was the parent, kept this as parent. Easily accessible without issues with collision prevention
				ipParentStation := ipEachMover.CurrentTrack.StationAhedPosition(ipEachMover.PositionOnTrack);
				IF ipEachMover.LastValidParentStation = ipParentStation AND ipParentStation <> 0 THEN
					//Set as new parent
					ipParentStation.AddMoverToQueue(ipEachMover);
					CONTINUE; //Check next mover
				END_IF
				
				//Prio 2: If the station closest was the parent, +/- 10mm . Maybe mall issues with collision prevention
				ipParentStation := ipEachMover.CurrentTrack.StationClosestTo(ipEachMover.PositionOnTrack);
				fDistToStation := F_DistXYVectors(ipParentStation.PositionOnTrackXYZABC, ipEachMover.PositionSet);
				IF ipEachMover.LastValidParentStation = ipParentStation AND ipParentStation <> 0 AND fDistToStation < 10.0 THEN
					//Set as new parent
					ipParentStation.AddMoverToQueue(ipEachMover);
					CONTINUE; //Check next mover
				END_IF
				
				//Prio 3: Get any station ahead current position
				ipParentStation := ipEachMover.CurrentTrack.StationAhedPosition(ipEachMover.PositionOnTrack);
				//Set as new parent
				ipParentStation.AddMoverToQueue(ipEachMover);
			END_IF
		END_WHILE
		THIS^.fbMoversPresent.RestoreIterator();	
	
		nSeqJoiningStation := 30;	
	
	
	
	30: //Send Movers to parent - shortest way
		THIS^.fbMoversPresent.ResetIterator();
		WHILE THIS^.fbMoversPresent.HasNextObject() DO
			//Do for all Movers whitout a target station
			IF ToXpMover(THIS^.fbMoversPresent.GetNextObject(),ipEachMover) AND_THEN (ipEachMover.ParentStation <> 0) AND_THEN __QUERYINTERFACE(ipEachMover,ipEachMoverPlc) THEN
				//Set Path dynamic constraint to settings in XPlanarParameterlist. 0=Defalt
				IF XPlanarParameterlist.F_ENABLING_ON_TRACK_VELOCITY <> 0 THEN fVelo := XPlanarParameterlist.F_ENABLING_ON_TRACK_VELOCITY;END_IF
				IF XPlanarParameterlist.F_ENABLING_ON_TRACK_ACC_DEC <> 0 THEN fAccDec := XPlanarParameterlist.F_ENABLING_ON_TRACK_ACC_DEC;END_IF
			
				//Increase or decrease the mover DynConstraint for approaching the station 
				ipEachMoverPlc.SetDynConstraint_Path(	V:= fVelo, 
														A:= fAccDec, 
														D:= fAccDec, 
														J:= Tc3_Mc3Definitions.MC_DEFAULT);
		
				// gap depending on current position
				fCalcualtedGapAtMoverPosition := ipEachMover.CurrentTrack.GapAtPosition(ipEachMover.PositionOnTrack);
		
				hr := GetMostSignificant(hr, ipEachMover.MoveOnTrack_ShortestWay(ipTrack := ipEachMover.ParentStation.AccocietedTrack,
																				fPosition := ipEachMover.ParentStation.PositionOnTrack, 
																				fGap := fCalcualtedGapAtMoverPosition));
				
					
				END_IF
		END_WHILE
		THIS^.fbMoversPresent.RestoreIterator();		

		IF CheckOk(hr) THEN 
			nSeqJoiningStation := 100;
		ELSIF FAILED(hr) THEN
			nSeqJoiningStation := 1000 + nSeqJoiningStation;
		END_IF	
	
	
		
	100: //Delay to allow the movers to start movement
		fbDelayJoiningStation.IN := TRUE;
		fbDelayJoiningStation.PT := T#100MS;
		IF fbDelayJoiningStation.Q THEN
			nSeqJoiningStation := 110;
			fbDelayJoiningStation.IN := FALSE;
		END_IF
	
	
	110: //Wait for all movers until the movement is completed(speed =0)
		THIS^.fbMoversPresent.ResetIterator();
		WHILE THIS^.fbMoversPresent.HasNextObject() DO
			IF ToXpMover(THIS^.fbMoversPresent.GetNextObject(),ipEachMover) THEN
				//Check all movers if an error is active
				IF ipEachMover.Feedback.Error THEN
					hr := GetMostSignificant(hr, ipEachMover.Feedback.HR);
				//Wait for all movers to stop/finish movement
				ELSIF NOT (ipEachMover.Standstill) THEN
					hr := GetMostSignificant(hr, S_PENDING);
				END_IF
			END_IF
		END_WHILE 
		THIS^.fbMoversPresent.RestoreIterator();
		
		IF CheckOk(hr) THEN 
			nSeqJoiningStation := 500;
		ELSIF FAILED(hr) THEN
			nSeqJoiningStation := 1000 + nSeqJoiningStation;
		END_IF			

		
	500: // Check if a mover passes his parent station and is not abel to drive backwarts due to CA
		(* every mover who has not made it to his target position (presumably because of CA) gets a new parent station which is definitely in front and can therefore be reached.
			Blocked movers are thus released. This should have no effect on all other movers as the parent remains identical. *)
		
		//Empty Mover queue in station
		THIS^.fbStationsUsed.ResetIterator();
		WHILE THIS^.fbStationsUsed.HasNextObject() DO
			IF __QUERYINTERFACE(THIS^.fbStationsUsed.GetNextObject(), ipEachStation) THEN
				ipEachStation.DeleteMoversQueue(); // This is also reset the parent of each mover
			END_IF
		END_WHILE
		THIS^.fbStationsUsed.RestoreIterator();

		//Set first station ahead as target or set again last valide station
		THIS^.fbMoversPresent.ResetIterator();
		WHILE THIS^.fbMoversPresent.HasNextObject() DO
			IF ToXpMover(THIS^.fbMoversPresent.GetNextObject(),ipEachMover) THEN
				refPosition REF= ipEachMover.LastValidParentStation.PositionOnTrackXYZABC;
				bMoverAtCmdPos := F_DistXYVectors(ipEachMover.PositionSet, refPosition) < 1.0;
				//Set again last parent
				IF bMoverAtCmdPos THEN
					ipEachMover.LastValidParentStation.AddMoverToQueue(ipEachMover);
				ELSE
					ipParentStation := ipEachMover.CurrentTrack.StationAhedPosition(ipEachMover.PositionOnTrack);
					ipParentStation.AddMoverToQueue(ipEachMover);
				END_IF
			END_IF
		END_WHILE 
		THIS^.fbMoversPresent.RestoreIterator();
		nSeqJoiningStation := 501;
		
		
	501: //Start movement - shortest way
		THIS^.fbMoversPresent.ResetIterator();
		WHILE THIS^.fbMoversPresent.HasNextObject() DO
			//Do for all Movers whitout a target station
			IF ToXpMover(THIS^.fbMoversPresent.GetNextObject(),ipEachMover) AND_THEN (ipEachMover.ParentStation <> 0) AND_THEN __QUERYINTERFACE(ipEachMover,ipEachMoverPlc) THEN
				//Set Path dynamic constraint to settings in XPlanarParameterlist. 0=Defalt
				IF XPlanarParameterlist.F_ENABLING_ON_TRACK_VELOCITY <> 0 THEN fVelo := XPlanarParameterlist.F_ENABLING_ON_TRACK_VELOCITY;END_IF
				IF XPlanarParameterlist.F_ENABLING_ON_TRACK_ACC_DEC <> 0 THEN fAccDec := XPlanarParameterlist.F_ENABLING_ON_TRACK_ACC_DEC;END_IF
			
				//Increase or decrease the mover DynConstraint for approaching the station 
				ipEachMoverPlc.SetDynConstraint_Path(	V:= fVelo, 
														A:= fAccDec, 
														D:= fAccDec, 
														J:= Tc3_Mc3Definitions.MC_DEFAULT);
		
				// gap depending on current position
				fCalcualtedGapAtMoverPosition := ipEachMover.CurrentTrack.GapAtPosition(ipEachMover.PositionOnTrack);
		
				hr := GetMostSignificant(hr, ipEachMover.MoveOnTrack_ShortestWay(ipTrack := ipEachMover.ParentStation.AccocietedTrack,
																				fPosition := ipEachMover.ParentStation.PositionOnTrack, 
																				fGap := fCalcualtedGapAtMoverPosition));
				
					
				END_IF
		END_WHILE
		THIS^.fbMoversPresent.RestoreIterator();		

		IF CheckOk(hr) THEN 
			nSeqJoiningStation := SEQ_DONE;
		ELSIF FAILED(hr) THEN
			nSeqJoiningStation := 1000 + nSeqJoiningStation;
		END_IF	

	SEQ_DONE:
		;
	
	1000..1999://Error
		hr := GetMostSignificant(hr, E_FAIL);
END_CASE

//Update
fbDelayJoiningStation();


//Return value
IF FAILED(hr) THEN 
	//Error
    JoiningStation := GetMostSignificant(hr, E_FAIL);
ELSIF (nSeqJoiningStation = SEQ_DONE) THEN
	//Done
    JoiningStation := S_OK;
ELSE
	//Busy
    JoiningStation := S_PENDING;;
END_IF
END_METHOD

METHOD PROTECTED JoiningTrack : HRESULT
VAR	
	hr : HRESULT;
	ipClosestTrack, ipLastTrack : I_XP_Track;	
	ipEachMover : I_XP_Mover;
	ipEachTrack : I_XP_Track;
	fDistance : LREAL;
	fShortestDistance : LREAL;
	fDistToLastValidPos : LREAL;
	bUseClosestTrack : BOOL;
END_VAR
CASE nSeqJoiningTrack OF

	0: //Init
		IF fbTracks.IsEmpty THEN
			nSeqJoiningTrack := SEQ_DONE;
		ELSE
			nSeqJoiningTrack := 10;
		END_IF

		
	10: //Last or Closest Track	
		//compare to the last valid position whether the mover is still unchanged on the tile. 
		//If there is only a small movement <5mm, an attempt is made to move to the last position. 
		//Otherwise the closest track is moved to
		THIS^.fbMoversPresent.ResetIterator();
		WHILE THIS^.fbMoversPresent.HasNextObject() DO
			IF ToXpMover(THIS^.fbMoversPresent.GetNextObject(),ipEachMover) THEN
				//Calculate distance
				fDistToLastValidPos := F_DistXYVectors(ipEachMover.LastValidPositionXYZABC, ipEachMover.PositionSet);
	
				IF fDistToLastValidPos > 5.0 OR ipEachMover.LastValidTrack = 0 THEN
					bUseClosestTrack := TRUE;
					EXIT;
				END_IF
	
			END_IF
		END_WHILE
		THIS^.fbMoversPresent.RestoreIterator();	
		
		
		IF bUseClosestTrack THEN
			//Closest
			nSeqJoiningTrack := 50;
		ELSE
			//Last
			nSeqJoiningTrack := 60;
		END_IF
		
		
		
	50:// Join closest track
		THIS^.fbMoversPresent.ResetIterator();
		WHILE THIS^.fbMoversPresent.HasNextObject() DO
			IF ToXpMover(THIS^.fbMoversPresent.GetNextObject(),ipEachMover) THEN
				
				//check all track to decide which is the closest
				//start with the greatest possible distance, so that each track is definitely closer
				fShortestDistance := CHALET_BaseComponents.GVL_Datatypes.cMaxLreal; 
				THIS^.fbTracks.ResetIterator();			
				WHILE THIS^.fbTracks.HasNextObject() DO
					IF ToXpTrack(THIS^.fbTracks.GetNextObject(),ipEachTrack) THEN
						fDistance := ipEachMover.DistToTrack(ipEachTrack);
						//closer track found
						IF fDistance <= fShortestDistance THEN
							ipClosestTrack := ipEachTrack;
							fShortestDistance := fDistance;
						END_IF
					END_IF
				END_WHILE
				THIS^.fbTracks.RestoreIterator();		
				

				IF ipClosestTrack <> 0 THEN
					hr := GetMostSignificant(hr, ipEachMover.JoinTrack(ipClosestTrack));
				ELSE
					hr := GetMostSignificant(hr, E_FAIL);
				END_IF
			
				
			END_IF
		END_WHILE
		THIS^.fbMoversPresent.RestoreIterator();
		nSeqJoiningTrack := 100;		
		
		
	60:// Move to last known position
		THIS^.fbMoversPresent.ResetIterator();
		WHILE THIS^.fbMoversPresent.HasNextObject() DO
			IF ToXpMover(THIS^.fbMoversPresent.GetNextObject(),ipEachMover) THEN
				hr := GetMostSignificant(hr, ipEachMover.MoveXY(ipEachMover.LastValidPositionXYZABC.x, ipEachMover.LastValidPositionXYZABC.y));
			END_IF
		END_WHILE
		THIS^.fbMoversPresent.RestoreIterator();
		nSeqJoiningTrack := 61;		
		
	61: // Moving check feedback
		THIS^.fbMoversPresent.ResetIterator();
		WHILE THIS^.fbMoversPresent.HasNextObject() DO
			IF ToXpMover(THIS^.fbMoversPresent.GetNextObject(),ipEachMover) THEN
				// Check mover errors
				hr := GetMostSignificant(hr, ipEachMover.Feedback.HR);
			END_IF
		END_WHILE
		THIS^.fbMoversPresent.RestoreIterator();		
		
		IF CheckOk(hr) THEN 
			nSeqJoiningTrack := 62;
		ELSIF FAILED(hr) THEN
			nSeqJoiningTrack := 1000 + nSeqJoiningTrack;
		END_IF	
		
	62: //Join last valid track
		THIS^.fbMoversPresent.ResetIterator();
		WHILE THIS^.fbMoversPresent.HasNextObject() DO
			IF ToXpMover(THIS^.fbMoversPresent.GetNextObject(),ipEachMover) THEN
				ipLastTrack := ipEachMover.LastValidTrack;
				hr := GetMostSignificant(hr, ipEachMover.JoinTrack(ipLastTrack));
			END_IF
		END_WHILE
		THIS^.fbMoversPresent.RestoreIterator();
		nSeqJoiningTrack := 100;
		
		
	100: // Joining  track check feedback
		THIS^.fbMoversPresent.ResetIterator();
		WHILE THIS^.fbMoversPresent.HasNextObject() DO
			IF ToXpMover(THIS^.fbMoversPresent.GetNextObject(),ipEachMover) THEN
				
				// Check mover errors
				hr := GetMostSignificant(hr, ipEachMover.Feedback.HR);
				
				//Check if Mover is on track
				IF NOT (ipEachMover.Mode = MC_PLANAR_MOVER_COMMAND_MODE.OnTrack) THEN
					hr := GetMostSignificant(hr, S_PENDING);
				END_IF
			END_IF
		END_WHILE
		THIS^.fbMoversPresent.RestoreIterator();
		
		IF CheckOk(hr) THEN 
			nSeqJoiningTrack := SEQ_DONE;
		ELSIF FAILED(hr) THEN
			nSeqJoiningTrack := 1000 + nSeqJoiningTrack;
		END_IF			

		
	1000..1999://Error
		hr := GetMostSignificant(hr, E_FAIL);
END_CASE

		
		
//Return value
IF FAILED(hr) THEN 
	//Error
    JoiningTrack := GetMostSignificant(hr, E_FAIL);
ELSIF (nSeqJoiningTrack = SEQ_DONE) THEN
	//Done
    JoiningTrack := S_OK;
ELSE
	//Busy
    JoiningTrack := S_PENDING;;
END_IF
END_METHOD

METHOD Disable : I_CH_Feedback
VAR_INPUT
END_VAR
//Disable is allways posible, but only if not already active
IF THIS^.nSeqDisabling = 0 OR THIS^.nSeqDisabling >= SEQ_DONE THEN
	THIS^.nSeqDisabling 	:= 1;
	THIS^.nSeqEnabling 		:= 0;
	
	THIS^.eActiveCommand 					:= CHALET_NC.E_NcAxisCommands.Disable;
	THIS^.fbFeedback.ActiveCommand 			:= TO_STRING(THIS^.eActiveCommand);	
	THIS^.fbFeedback.LastCommandAccepted	:= TRUE;		
	THIS^.fbFeedback.Busy 					:= TRUE;
			
	
ELSE
	THIS^.fbFeedback.LastCommandAccepted	:= FALSE;	
END_IF

Disable := THIS^.fbFeedback;
END_METHOD

{attribute 'monitoring':='call'}
PROPERTY Disabled : BOOL
GET
Disabled := nSeqDisabling = SEQ_DONE OR 
			(nSeqDisabling = 0 AND nSeqEnabling = 0);
END_GET
END_PROPERTY

METHOD PROTECTED Disabling : HRESULT
VAR
	hr : HRESULT;
	bOk : BOOL := TRUE;
	ipEachMover : I_XP_Mover;
	ipEachTrack : I_XP_Track;
	ipEachStation : I_XP_Station;
END_VAR
VAR_INST
	hrLastCycle : HRESULT;
END_VAR
Disabling := S_PENDING;
CASE nSeqDisabling OF
	0: // Idle
		Disabling := S_OK;
		
		
	1: // Halt movers - keep at first position for a fast stop reaction
		THIS^.fbMoversPresent.ResetIterator();
		WHILE THIS^.fbMoversPresent.HasNextObject() DO
			IF ToXpMover(THIS^.fbMoversPresent.GetNextObject(),ipEachMover) THEN
				IF XPlanarParameterlist.B_QUICKSTOP_ON_DISABLING THEN
					//The mover stops immediately at the current position
					hr := GetMostSignificant(hr, ipEachMover.Disable());
				ELSE
					//The mover cancels the superimposed ExternalSetpoint movement and returns to the track with maximum dynamic. -> Like a rubber band
					hr := GetMostSignificant(hr, ipEachMover.Halt());
				END_IF
			END_IF
		END_WHILE
		THIS^.fbMoversPresent.RestoreIterator();
	    		
		IF CheckOk(hr) THEN 
			nSeqDisabling := 20;
		ELSE
			nSeqDisabling := 1000 + nSeqDisabling;
		END_IF	
	
		
	20: // Halting movers
		THIS^.fbMoversPresent.ResetIterator();
		WHILE THIS^.fbMoversPresent.HasNextObject() DO
			IF ToXpMover(THIS^.fbMoversPresent.GetNextObject(),ipEachMover) THEN
				bOk := bOk AND ipEachMover.Standstill;
			END_IF
		END_WHILE
		THIS^.fbMoversPresent.RestoreIterator();
		
		IF bOk THEN 
			nSeqDisabling := 30;
		END_IF	
			
		
	
	30: // Reset movers
		THIS^.fbMoversPresent.ResetIterator();
		WHILE THIS^.fbMoversPresent.HasNextObject() DO
			IF ToXpMover(THIS^.fbMoversPresent.GetNextObject(),ipEachMover) THEN
				hr := GetMostSignificant(hr, ipEachMover.Reset());
			END_IF
		END_WHILE
		
		IF CheckOk(hr) THEN 
			nSeqDisabling := 40;
		ELSE
			nSeqDisabling := 1000 + nSeqDisabling;
		END_IF		
		
		
	40: // Resetting movers
		THIS^.fbMoversPresent.ResetIterator();
		WHILE THIS^.fbMoversPresent.HasNextObject() DO
			IF ToXpMover(THIS^.fbMoversPresent.GetNextObject(),ipEachMover) THEN
				hr := GetMostSignificant(hr, ipEachMover.Feedback.HR);
			END_IF
		END_WHILE
		
		IF CheckOk(hr) THEN 
		//	nSeqDisabling := 45;
			nSeqDisabling := 50;
		ELSIF FAILED(hr) THEN
			nSeqDisabling := 1000 + nSeqDisabling;
		END_IF
		
		
		
(*		
	45: // Stop external Setpoint 
		THIS^.fbMovers.ResetIterator();
		WHILE THIS^.fbMovers.HasNextObject() DO
			IF ToXpMover(THIS^.fbMovers.GetNextObject(),iTempMover) THEN
				hr := GetMostSignificant(hr, iTempMover.StopExternalSetpoint());
			END_IF
		END_WHILE
		
		IF CheckOk(hr) THEN 
			nSeqDisabling := 46;
		ELSE
			nSeqDisabling := 1000 + nSeqDisabling;
		END_IF			
		

	46: // Stoping external Setpoint 
		THIS^.fbMovers.ResetIterator();
		WHILE THIS^.fbMovers.HasNextObject() DO
			IF ToXpMover(THIS^.fbMovers.GetNextObject(),iTempMover) THEN
				hr := GetMostSignificant(hr, iTempMover.Feedback.HR);
			END_IF
		END_WHILE
		
		IF CheckOk(hr) THEN 
			nSeqDisabling := 50;
		ELSIF FAILED(hr) THEN
			nSeqDisabling := 1000 + nSeqDisabling;
		END_IF			
*)		
		
		
		
	50: // Disable movers
		THIS^.fbMoversPresent.ResetIterator();
		WHILE THIS^.fbMoversPresent.HasNextObject() DO
			IF ToXpMover(THIS^.fbMoversPresent.GetNextObject(),ipEachMover) THEN
				hr := GetMostSignificant(hr, ipEachMover.Disable());
			END_IF
		END_WHILE
		
		IF CheckOk(hr) THEN 
			nSeqDisabling := 60;
		ELSE
			nSeqDisabling := 1000 + nSeqDisabling;
		END_IF			
		

		
	60: // Disabling movers
		THIS^.fbMoversPresent.ResetIterator();
		WHILE THIS^.fbMoversPresent.HasNextObject() DO
			IF ToXpMover(THIS^.fbMoversPresent.GetNextObject(),ipEachMover) THEN
				hr := GetMostSignificant(hr, ipEachMover.Feedback.HR);
			END_IF
		END_WHILE
		
		IF CheckOk(hr) THEN 
			nSeqDisabling := 61;
		ELSIF FAILED(hr) THEN
			nSeqDisabling := 1000 + nSeqDisabling;
		END_IF		


	61: // Reset track
		THIS^.fbTracks.ResetIterator();
		WHILE THIS^.fbTracks.HasNextObject() DO
			IF ToXpTrack(THIS^.fbTracks.GetNextObject(),ipEachTrack) THEN
				hr := GetMostSignificant(hr, ipEachTrack.Reset());
			END_IF
		END_WHILE
		
		IF CheckOk(hr) THEN 
			nSeqDisabling := 62;
		ELSE
			nSeqDisabling := 1000 + nSeqDisabling;
		END_IF		
		
		
	62: // Resetting track
		THIS^.fbTracks.ResetIterator();
		WHILE THIS^.fbTracks.HasNextObject() DO
			IF ToXpTrack(THIS^.fbTracks.GetNextObject(),ipEachTrack) THEN
				hr := GetMostSignificant(hr, ipEachTrack.Feedback.HR);
			END_IF
		END_WHILE
		
		IF CheckOk(hr) THEN 
			nSeqDisabling := 63;
		ELSIF FAILED(hr) THEN
			nSeqDisabling := 1000 + nSeqDisabling;
		END_IF	

				
	63: // Reset group
		hr := ipGroup.Reset();
		
		IF CheckOk(hr) THEN 
			nSeqDisabling := 64;
		ELSE
			nSeqDisabling := 1000 + nSeqDisabling;
		END_IF		
		
		
	64: // Resetting group
		hr := ipGroup.Feedback.HR;
		
		IF CheckOk(hr) THEN 
			nSeqDisabling := 70;
		ELSIF FAILED(hr) THEN
			nSeqDisabling := 1000 + nSeqDisabling;
		END_IF		
		
		
		

   70: // Disable tracks
		THIS^.fbTracks.ResetIterator();
		WHILE THIS^.fbTracks.HasNextObject() DO
			IF ToXpTrack(THIS^.fbTracks.GetNextObject(),ipEachTrack) THEN
				hr := GetMostSignificant(hr, ipEachTrack.Disable());
			END_IF
		END_WHILE
		
		IF CheckOk(hr) THEN 
			nSeqDisabling := 80;
		ELSE
			nSeqDisabling := 1000 + nSeqDisabling;
		END_IF			
   
		
   80: // Disabling tracks
		THIS^.fbTracks.ResetIterator();
		WHILE THIS^.fbTracks.HasNextObject() DO
			IF ToXpTrack(THIS^.fbTracks.GetNextObject(),ipEachTrack) THEN
				hr := GetMostSignificant(hr, ipEachTrack.Feedback.HR);
			END_IF
		END_WHILE
		
		IF CheckOk(hr) THEN 
			nSeqDisabling := 90;
		ELSIF FAILED(hr) THEN
			nSeqDisabling := 1000 + nSeqDisabling;
		END_IF	
				

	90: // Disable group
		hr := ipGroup.Disable();
		
		IF CheckOk(hr) THEN 
			nSeqDisabling := 100;
		ELSE
			nSeqDisabling := 1000 + nSeqDisabling;
		END_IF	
		
		
   100: // Disabling group
		hr := ipGroup.Feedback.HR;
		
		IF CheckOk(hr) THEN 
			nSeqDisabling := 102;
		ELSIF FAILED(hr) THEN
			nSeqDisabling := 1000 + nSeqDisabling;
		END_IF	

		
	102: //Delete all paths. These are only temporary objects and will be recreated the next time they are enabled
		THIS^.fbStationsUsed.ResetIterator();
		WHILE THIS^.fbStationsUsed.HasNextObject() DO
			IF ToXpStation(THIS^.fbStationsUsed.GetNextObject(),ipEachStation) THEN
				hr := ipEachStation.Disassemble();
			END_IF
		END_WHILE
	
		IF CheckOk(hr) THEN 
			nSeqDisabling := 103;
		ELSE
			nSeqDisabling := 1000 + nSeqDisabling;
		END_IF			
		
		
	103: //Delete all paths. These are only temporary objects and will be recreated the next time they are enabled
		THIS^.fbListAllMovers.ResetIterator();
		WHILE THIS^.fbListAllMovers.HasNextObject() DO
			IF ToXpMover(THIS^.fbListAllMovers.GetNextObject(),ipEachMover) THEN
				hr := ipEachMover.Disassemble();
			END_IF
		END_WHILE
	
		IF CheckOk(hr) THEN 
			nSeqDisabling := 105;
		ELSE
			nSeqDisabling := 1000 + nSeqDisabling;
		END_IF		
		
		
		
		
		
  105: // Remove tracks from group
		THIS^.fbTracks.ResetIterator();
		WHILE THIS^.fbTracks.HasNextObject() DO
			IF ToXpTrack(THIS^.fbTracks.GetNextObject(),ipEachTrack) THEN
				hr := GetMostSignificant(hr, ipEachTrack.RemoveFromGroup());
			END_IF
		END_WHILE
		
		IF CheckOk(hr) THEN 
			nSeqDisabling := 106;
		ELSE
			nSeqDisabling := 1000 + nSeqDisabling;
		END_IF			
   
		
   106: // Removing tracks from group
		THIS^.fbTracks.ResetIterator();
		WHILE THIS^.fbTracks.HasNextObject() DO
			IF ToXpTrack(THIS^.fbTracks.GetNextObject(),ipEachTrack) THEN
				bOk := bOk AND ipEachTrack.PlanarTrack.MCTOPLC_STD.GroupOID = 0;
			END_IF
		END_WHILE
		
		IF bOk THEN 
			nSeqDisabling := 110;
		END_IF	
		
		
	110: // Remove movers from group
		THIS^.fbMoversPresent.ResetIterator();
		WHILE THIS^.fbMoversPresent.HasNextObject() DO
			IF ToXpMover(THIS^.fbMoversPresent.GetNextObject(),ipEachMover) THEN
				hr := GetMostSignificant(hr, ipEachMover.RemoveFromGroup());
			END_IF
		END_WHILE
		
		IF CheckOk(hr) THEN 
			nSeqDisabling := 120;
		ELSE
			nSeqDisabling := 1000 + nSeqDisabling;
		END_IF		
	
		
	120: // Removing movers from group
		THIS^.fbMoversPresent.ResetIterator();
		WHILE THIS^.fbMoversPresent.HasNextObject() DO
			IF ToXpMover(THIS^.fbMoversPresent.GetNextObject(),ipEachMover) THEN
				bOk := bOk AND ipEachMover.PlanarMover.MCTOPLC.STD.GroupOID = 0;
			END_IF
		END_WHILE
		
		IF bOk THEN 
			nSeqDisabling := 130;
		END_IF		
	
		
	130: // Remove envirement from group
		hr := ipEnvironment.RemoveFromGroup();
		
		IF CheckOk(hr) THEN 
			nSeqDisabling := 140;
		ELSE
			nSeqDisabling := 1000 + nSeqDisabling;
		END_IF		
		
		
   140: // Removing envirement from group
		hr := ipEnvironment.Feedback.HR;
	
		IF CheckOk(hr) THEN 
			nSeqDisabling := 200;
		ELSIF FAILED(hr) THEN
			nSeqDisabling := 1000 + nSeqDisabling;
		END_IF			
		
		
   200: // Reset Utility errors
		ipEnvironment.UtilityEnvirement.ErrorAcknowledge();
		nSeqDisabling := SEQ_DONE;

		
	
   SEQ_DONE: //Done
   		Disabling := S_OK;

		
	1000..1999://Error
		hr := GetMostSignificant(hrLastCycle, E_FAIL);
	
END_CASE

//store last information
hrLastCycle := hr;

// Propagate error
IF FAILED(hr) THEN
	Disabling := hr;
END_IF
END_METHOD

METHOD Enable : CHALET_BaseComponents.I_CH_Feedback
VAR_INPUT
END_VAR
IF NOT THIS^.fbFeedback.Done THEN
	//Error active/not ready
	THIS^.fbFeedback.LastCommandAccepted 	:= FALSE;

ELSIF nSeqEnabling <> 0 THEN
	//System is partial or full enabled. Disable first.
	THIS^.fbFeedback.LastCommandAccepted 	:= FALSE;
ELSE
	THIS^.nSeqDisabling 	:= 0;
	THIS^.nSeqEnabling 		:= 1;
	
	THIS^.eActiveCommand 				:= CHALET_NC.E_NcAxisCommands.Enable;
	THIS^.fbFeedback.ActiveCommand 		:= TO_STRING(THIS^.eActiveCommand);	
	THIS^.fbFeedback.LastCommandAccepted:= TRUE;		
	THIS^.fbFeedback.Busy 				:= TRUE;	
END_IF

Enable := THIS^.fbFeedback;
END_METHOD

{attribute 'monitoring':='call'}
PROPERTY Enabled : BOOL
GET
Enabled := nSeqEnabling = SEQ_DONE;
END_GET
END_PROPERTY

METHOD PROTECTED Enabling : HRESULT
VAR

	hr : HRESULT;
	bWatchDogActive : BOOL;
	ipTempMover : I_XP_Mover;
	ipTempMoverPlc : I_XP_Mover_PLC;
	ipTempStation : I_XP_Station;
	ipTempTrack : I_XP_Track;
	stController : ST_TcIoControllersOn;
	lrCRotationShortestPos : LREAL;
	bOk : BOOL;
	nSupSeq : UINT;
	nIdx : UINT;
	sMoverType : STRING;
	fDistLastToSet : LREAL;
	fMaxError : LREAL;
	nMoversDetected, nMoverExpected : UDINT;
	bMoverIsMissing : BOOL;
	eMoverDetectionStatus : MoverDetectionStatus;
	stCoordMoverCommStatus : CoordinatedMoverCommStatus;
	ipMoverTComObject : ITComObject;
	nParaSize : UDINT;
	pParaData : PVOID;
	eAccessory : MoverAccessoryID;//(APM9000_0000:=0, APM9001_0000:=1)
END_VAR

VAR_INST
	{attribute 'hide'}	
	fbTimeOutSeq : TON; 
	{attribute 'hide'}	
	hrLastCycle 	: HRESULT;
	{attribute 'hide'}	
	nlastState	: UINT;
	
	// todo hide
	bIdBumperOnAllMovers : BOOL;
	
	{attribute 'hide'}	
	fbTimeOutEnabling : FB_TcAlarm;
	{attribute 'hide'}	
	fbErrorEnabling : FB_TcAlarm;
	{attribute 'hide'}	
	fbErrorMoverDetection : FB_TcAlarm;
	{attribute 'hide'}	
	bAllMoverOrientationValide : BOOL;	
	{attribute 'hide'}	
	bAllMoverIdDetectionValide : BOOL;
END_VAR
Enabling := S_PENDING;
CASE nSeqEnabling OF
	0: // Idle
		Enabling := S_OK;	
				
	1: // Prepare 
		THIS^.fbListAllMovers.Clear();
		THIS^.fbListAllMovers.AddList(THIS^.fbMoversPresent);
		THIS^.fbListAllMovers.AddList(THIS^.fbMoversNotPresent);
		
		
